/// Returns last zone index that can be found between start and end position, direction according windows ascending
/// REMARK: Size of area to be checked has influence to performance of method
METHOD M_GetLastZoneIndex : UINT // Returns ZoneIndex > 0, otherwise 0
VAR_INPUT
	mAbsoluteStartPosition	: UDINT; // Start position on the tracking [mm]
	mAbsoluteEndPosition	: UDINT; // End position on the tracking [mm]
	mOnlyZonesWithTU		: BOOL; // Check only zones with physical TU
END_VAR
END_METHOD

/// Searches through all available zones and add all zone index of ActionId to pData
/// Remark: Amount of available zones has influence to performance.
/// Remark: Existing entries in pData get overwritten.
METHOD M_GetPendingAssignments : BOOL // Returns true if all found zones could be added to pData, otherwise false
VAR_INPUT
	mActionId				: INT; // ID of action which requests zone (<>0)
	mpData 					: POINTER TO UINT; // Address of Value or Array to store the result
	mDataLen				: UINT; // Size of data
END_VAR
VAR_OUTPUT
	mCount					: UINT; // Number of entries added to pData
END_VAR
END_METHOD

/// Converts an absolute position into the current position on the tracking
METHOD M_GetTrackingPosition : UDINT // Converted position on tracking [mm]
VAR_INPUT
	mAbsolutePosition	: UDINT; // Absolute position 
END_VAR
END_METHOD

/// Returns TU end position of a zone on tracked distance
/// Remark: When no TU available the return value is 0, but is notfied with output "NoTuAvailable"
METHOD M_GetTU_EndPosition : UDINT // Returns position of TU end [mm]
VAR_INPUT
	mZoneIndex			: UINT; // Index of zone
END_VAR
VAR_OUTPUT
	mNoTU_Available		: BOOL; // No TU Available
END_VAR
END_METHOD

/// Returns TU start position of a zone on tracked distance
/// Remark: When no TU available the return value is 0, but is notfied with output "NoTuAvailable"
METHOD M_GetTU_StartPosition : UDINT // Start position of TU [mm]
VAR_INPUT
	mZoneIndex			: UINT; // Index of zone
END_VAR
VAR_OUTPUT
	mNoTU_Available		: BOOL; // No TU Available
END_VAR
END_METHOD

/// Returns position of Zone end on tracked distance
METHOD M_GetZoneEndPosition : UDINT // Position of Zone end [mm]
VAR_INPUT
	mZoneIndex			: UINT; // Index of zone
END_VAR
END_METHOD

/// Returns ZoneIndex at AbsolutePosition
METHOD M_GetZoneIndex : UINT // Returns ZoneIndex > 0, otherwise 0
VAR_INPUT
	mAbsolutePosition	: UDINT; // Position on the tracking [mm]
END_VAR
END_METHOD

/// Returns position of Zone start on tracked distance
METHOD M_GetZoneStartPosition : UDINT // Position of Zone start [mm]
VAR_INPUT
	mZoneIndex			: UINT; // Index of zone
END_VAR
END_METHOD

/// Inhibits shifting on a specific zone
METHOD M_InhibitShifting : BOOL // Returns true if successfully, otherwise false (e.g. Zone not found or not in use)
VAR_INPUT
	mZoneIndex		: UINT; // Zone index
	mInhibit		: BOOL; // True = Inhibit shifting
END_VAR
END_METHOD

/// Checks if a TU or a part of it, is found in a certain range.
METHOD M_IsTU_InRange : BOOL; // Returns true if present, otherwise false
VAR_INPUT
	mZoneIndex				: UINT; // Tracking zone index
	mAbsoluteStartRange		: UDINT; // Start range position on the tracking [mm]
	mAbsoluteEndRange		: UDINT; // End range position on the tracking [mm]
END_VAR
END_METHOD

/// Returns if a physical TU is present at mAbsolutePosition
METHOD M_IsTU_Present : BOOL; // Returns true if present, otherwise false
VAR_INPUT
	mAbsolutePosition		: UDINT; // Absolute position on tracking length
END_VAR
END_METHOD

/// Checks if a zone or a part of it,  is found in a certain range.
METHOD M_IsZoneInRange : BOOL; // Returns true if zone is in range, otherwise false
VAR_INPUT
	mZoneIndex				: UINT; // Tracking zone index
	mAbsoluteStartRange		: UDINT; // Start range position on the tracking [mm]
	mAbsoluteEndRange		: UDINT; // End range position on the tracking [mm]
END_VAR
END_METHOD

/// This function synchronize only a Front edge to a specific position and calculates the new TU length.
/// Remark: Zone begin gets adjusted to new front edge position. Spare windows in front of front edge get removed.
/// Remark: If at absolute position no zone is found, it search to the left for next front edge
/// until "mMaxFrontEdgeDeviation" to find one to synchronize.
METHOD M_ResyncOnlyFE : UINT // Returns > 0 of the synchronized Zone index, otherwise 0 (e.g. No Zone, No occupied zone)
VAR_INPUT
	mAbsolutePosition		: UDINT; // Absolute position [mm]
	mMaxFrontEdgeDeviation 	: UDINT; (* When zone can not be found at "Absolute position",
										a search upwards is executed to a limit of MaxFrontEdgeDeviation [mm]*)
END_VAR
END_METHOD

/// This function synchronize only Rear edge to a specific position and calculates new TU length.
/// Remark: Zone end gets adjusted to new rear edge position. Spare windows after rear edge get removed.
/// Remark: If at absolute position no zone is found, it search to the right
/// until "mMaxFrontEdgeDeviation" to find one to synchronize.
METHOD M_ResyncOnlyRE : UINT // Returns > 0 of the synchronized Zone index, otherwise 0
VAR_INPUT
	mAbsolutePosition		: UDINT; // Absolute position [mm]
	mMaxRearEdgeDeviation 	: UDINT; (* When zone can not be found at "Absolute position",
										a search upwards is executed to a limit of MaxRearEdgeDeviation [mm]*)
END_VAR
END_METHOD

/// This function synchronize whole TU aligned by Front edge to a specific position.
/// Rear edge is adjusted automatically to keep the length of TU.
/// Remark: If at absolute position no zone is found, it search to the left
/// until "mMaxFrontEdgeDeviation" to find one to synchronize.
METHOD M_ResyncTU_FE : UINT // Returns > 0 of the synchronized Zone index, otherwise 0
VAR_INPUT
	mAbsolutePosition		: UDINT; // Absolute position [mm]
	mMaxFrontEdgeDeviation 	: UDINT; (* When zone can not be found at "Absolute position",
										a search upwards is executed to a limit of MaxFrontEdgeDeviation [mm]*)
END_VAR
END_METHOD

/// This function synchronize whole TU aligned by Rear edge to a specific position.
/// Front edge is adjusted automatically to keep the length of TU.
/// Remark: If at absolute position no zone is found, it search to the right
/// until "mMaxFrontEdgeDeviation" to find one to synchronize.
METHOD M_ResyncTU_RE : UINT // Returns > 0 of the synchronized Zone index, otherwise 0
VAR_INPUT
	mAbsolutePosition		: UDINT; // Absolute position [mm]
	mMaxRearEdgeDeviation 	: UDINT; (* When zone can not be found at "Absolute position",
										a search upwards is executed to a limit of MaxRearEdgeDeviation [mm]*)
END_VAR
END_METHOD

/// Enlarges a zone by given value to upstream direction
METHOD M_ShortenZone : BOOL
VAR_INPUT
	mZoneIndex 				: UINT; // Zone index to enlarge
	mReductionLength		: UINT; // Reduce existing zone by this length [mm]
	mShiftFrontEdge			: BOOL; // Shift front edge for reduction
END_VAR
END_METHOD

/// Returns currently available amount of TUs
PROPERTY P_TU_Count : INT
GET
END_GET
END_PROPERTY

/// Access to Window table  for read operations
/// Remark: User has to ensure that writing does not influence the process in a bad way.
{attribute 'suppress_wrn_C0410'}
PROPERTY P_WindowTable : REFERENCE TO ARRAY[1..WindowTracking.MAX_NUMBER_OF_WINDOWS] OF ST_WindowTrackingWindow;
GET
END_GET
END_PROPERTY

/// Returns currently available amount of Zones
PROPERTY P_ZoneCount : INT
GET
END_GET
END_PROPERTY

/// Access to Zone table  for read operations
/// Remark: User has to ensure that writing does not influence the process in a bad way.
{attribute 'suppress_wrn_C0410'}
PROPERTY P_ZoneTable : REFERENCE TO ARRAY[1..WindowTracking.MAX_NUMBER_OF_ZONES] OF ST_WindowTrackingZone;
GET
END_GET
END_PROPERTY

END_INTERFACE

// ---- 20_Product/30_Toolbox/17_WindowTracking/10_Core/02_ITFs/I_WindowTrackingListener.TcIO
/// Window tracking listener 
INTERFACE I_WindowTrackingListener EXTENDS __System.IQueryInterface

/// Shifting completed event
METHOD M_TrackingShiftingCompletedEvent
VAR_INPUT
	mAbsolutePosition		: UDINT; // Absolute shifting start position [mm]
	mDistance				: UDINT; // Distance [mm] to be shifted
	mWindowIndex			: UINT; // Absolute position as window index on tracking
	mWindowsToShift			: UINT; // Distance to be shifted in amount of windows
END_VAR
END_METHOD

/// Shifting initiated event
METHOD M_TrackingShiftingInitiatedEvent
VAR_INPUT
	mAbsolutePosition		: UDINT; // Absolute shifting start position [mm]
	mDistance				: UDINT; // Distance [mm] to be shifted
	mWindowIndex			: UINT; // Absolute position as window index on tracking
	mWindowsToShift			: UINT; // Distance to be shifted in amount of windows
END_VAR
END_METHOD

/// Window tracking allocated new zone
METHOD M_TrackingTU_AddedEvent
VAR_INPUT
	mTrackingZoneIndex	: UINT; // New Zone index 
	mTrackingZoneData	: ST_WindowTrackingZone; // Data of deleted zone
END_VAR
END_METHOD

/// Window tracking deleted this zone
METHOD M_TrackingTU_DeletedEvent
VAR_INPUT
	mTrackingZoneIndex	: UINT; // Deleted zone index
	mTrackingZoneData	: ST_WindowTrackingZone; // Data of deleted zone
END_VAR
END_METHOD

/// Window tracking allocated new zone
METHOD M_TrackingZoneAddedEvent
VAR_INPUT
	mTrackingZoneIndex	: UINT; // New Zone index 
	mTrackingZoneData	: ST_WindowTrackingZone; // Data of deleted zone
END_VAR
END_METHOD

/// Window tracking deleted this zone
METHOD M_TrackingZoneDeletedEvent
VAR_INPUT
	mTrackingZoneIndex	: UINT; // Deleted zone index
	mTrackingZoneData	: ST_WindowTrackingZone; // Data of deleted zone
END_VAR
END_METHOD

/// A zone was enlarged event
METHOD M_TrackingZoneEnlargedEvent
VAR_INPUT
	mTrackingZoneIndex	: UINT; // Enlarged Zone index 
END_VAR
VAR_IN_OUT
	mOldTrackingZoneData : ST_WindowTrackingZone; // Zone data before modification
	mNewTrackingZoneData : ST_WindowTrackingZone; // Zone data after modification
END_VAR
END_METHOD

/// Window tracking moved this zone
METHOD M_TrackingZoneMovedEvent
VAR_INPUT
	mTrackingZoneIndex	: UINT; // Deleted zone index
	mTrackingZoneData	: ST_WindowTrackingZone; // Data of deleted zone
END_VAR
END_METHOD

/// A zone was shortened event
METHOD M_TrackingZoneShortenedEvent
VAR_INPUT
	mTrackingZoneIndex	: UINT; // Shortened Zone index 
END_VAR
VAR_IN_OUT
	mOldTrackingZoneData : ST_WindowTrackingZone; // Zone data before modification
	mNewTrackingZoneData : ST_WindowTrackingZone; // Zone data after modification
END_VAR
END_METHOD

END_INTERFACE

// ---- 20_Product/20_ProBox/MainProBox.TcPOU
PROGRAM MainProBox
(**************************************************************************************
 * 	Application		:	ProBox
 *	Revision		:	$$
 *	Revision date	:	$$
 *	Last changed by	:	$$
 *	URL				:	$$
 *
 *	Purpose			:	ProBox main application.
 *
 * ------------------------------------------------------------------------------------
 *	Copyright Swisslog [IP AG], Switzerland. All rights reserved.
 * 
 * ------------------------------------------------------------------------------------
 *	
 * 	Revision History: 
 *
 * 	VERSION			DATE			INITIALS			DESCRIPTION
 *	0.1				01.01.2001		swl					Example
 *
 **************************************************************************************)
VAR
	fbHardwareInputs					: FB_HardwareInputs;
	fbHardwareOutputs					: FB_HardwareOutputs;	
	fbSafetyCustomization				: FB_SafetyCompositionCustomized;
END_VAR
VAR_TEMP
BCFisInitiaded:BOOL;
		
END_VAR

 
(***************************************************************************************************************
  
***************************************************************************************************************)
BCFisInitiaded :=MainConv.Init;

EMULATION_ENABLED := TRUE;
IF(EMULATION_ENABLED) THEN
	MainConvEmulation();
END_IF

IF(BCFisInitiaded) THEN 
	IF(NOT EMULATION_ENABLED) THEN
		// Get HW Inputs
		fbHardwareInputs();
	END_IF		
	// run Custom debug functions
	F_DebugCompositionCustomization();  
END_IF
	
// Custom safety functions 
fbSafetyCustomization(_InitSafety:=BCFisInitiaded AND NOT EMULATION_ENABLED);
//run BCF
MainConv();

//if MainConv is initiated and not emulation enabled
IF(BCFisInitiaded) THEN
	//Set HW Outputs
	fbHardwareOutputs();		
END_IF

END_PROGRAM

// ---- 10_Project/10_App/11_Custom/FB_HardwareInputs.TcPOU
FUNCTION_BLOCK FB_HardwareInputs


;
// Example
(*
fbSG_001.HW_Inputs 								:= I_11_001_SG;
fbSG_001.HW_Inputs.ResetErrorPB 				:= I_11_001_SG.AutoOnPB;
fbSG_001.HW_Inputs.FeedbackMainContactorOFF[4] 	:= FALSE;
fbSG_001.HW_Inputs.EmergencyCircuitOK 			:= TRUE;
fbSG_001.HW_Inputs.MainContactorOFF 			:= I_11_001_SG.MainContactorOFF;

Main_Contactor_ON_Q := Main_Contactor_ON_I;
Main_Contactor_OFF_Q := Main_Contactor_OFF_I;
*)

END_FUNCTION_BLOCK

// ---- 10_Project/10_App/11_Custom/FB_HardwareOutputs.TcPOU
FUNCTION_BLOCK FB_HardwareOutputs


;
// Example
(*
Q_11_001_SG := fbSG_001.HW_Outputs;
Q_11_001_SG_Beacon_Error := fbSG_001.HW_Outputs.ErrorPending;
Q_11_001_SG_Beacon_Auto := fbSG_001.HW_Outputs.GroupStarted;
*)

END_FUNCTION_BLOCK

// ---- 10_Project/10_App/11_Custom/FB_SafetyCompositionCustomized.TcPOU
FUNCTION_BLOCK FB_SafetyCompositionCustomized
VAR_INPUT
	///true if initializing is active
	_InitSafety: BOOL;
END_VAR


IF(_InitSafety) Then
	//Add project specific safety code that shall execute during PLC init/reinit. 
	;
ELSE
	//Add project specific safety code here. 
	//renamed from Com_Error to FB_SafetyCompositionCustomized
	;
END_IF

END_FUNCTION_BLOCK

// ---- 20_Product/10_BCF/11_Conv/MainConv.TcPOU
PROGRAM MainConv
(**************************************************************************************
 * 	Application		:	BoxControl Framework
 *	Revision		:	$Revision: 404529 $
 *	Revision date	:	$Date: 2018-04-23 08:21:38 +0200 (Mo., 23 Apr 2018) $
 *	Last changed by	:	$Author: b7bolm $
 *	URL				:	$URL: http://almscdc.swisslog.com/repo/SWPD/Development/BoxControlFramework/20_Release/trunk/01_Software/BCF/BCF/JumpStart/20_Product/10_App/MainConv.TcPOU $
 *
 *	Purpose			:	Main program call.
 *
 * ------------------------------------------------------------------------------------
 *	Copyright Swisslog [IP AG], Switzerland. All rights reserved.
 * 
 * ------------------------------------------------------------------------------------
 *	
 * 	Revision History: 
 *
 * 	VERSION			DATE			INITIALS			DESCRIPTION
 *	0.1				01.01.2001		swl					Example
  *
 **************************************************************************************)
VAR
	Init								: BOOL := FALSE; // Application is initialized 
	
	ActivateSubsystemConfig				: BOOL; // Flag to activate the configuration of the Subsystem 
	ActivateGroupManagerConfig			: BOOL; // Flag to activate the configuration of the groupmanager 
	ActivateGroupConfig					: BOOL; // Flag to activate the configuration of the group 
	ActivatePositionConfig				: BOOL; // Flag to activate the configuration of the element 
	ActivateCommunicationConfig			: BOOL; // Flag to activate the configuration of the communication 
	
	InitializeSubsystem					: BOOL; // Flag to activate initialization
	InitializeGroupManager				: BOOL; // Flag to activate initialization
	InitializeGroups					: BOOL; // Flag to activate initialization
	InitializeFunctions					: BOOL; // Flag to activate initialization
	InitializeCommunication				: BOOL; // Flag to activate initialization
	InitializeElements					: BOOL; // Flag to activate initialization
	ReInit								: BOOL := TRUE; // Reinitialize application
	fbDebugMsg							: FB_DebugMsg; // Debug instance
	fbGetSystemTime						: GETSYSTEMTIME; // Gets the system time  
	LatchedTimeDW						: DWORD; // Latch the system time 
	LastTimeStamp						: DWORD; // Time stamp
	fbGetCurTaskIdx  					: GETCURTASKINDEX; // Returns the actual task index
	
	fbCommunicationComposition			: FB_CommunicationComposition; // Communication call
	fbElementComposition				: FB_ElementComposition; // Element calls
	fbElementCompositionCustomized		: FB_ElementCompositionCustomized; // Element calls
	fbFunctionComposition				: FB_FunctionComposition; // Function calls
	fbFunctionCompositionCustomized		: FB_FunctionCompositionCustomized; // Function calls
	fbGroupComposition					: FB_GroupComposition; // Group calls
	fbGroupCompositionCustomized		: FB_GroupCompositionCustomized; // Group calls
	fbSubsystemComposition				: FB_SubsystemComposition; // Subsystem calls
	fbSubsystemCompositionCustomized	: FB_SubsystemCompositionCustomized; // Subsystem calls
	fbDeleteOldTU_Data					: FB_DeleteOldTU_Data; // Checks old TU data
	SubsystemState						: ST_PositionState; // Subsystem state
END_VAR

// whow

(**************************************************************************************************************
   Update PLC data
***************************************************************************************************************)
A_UpdatePLC_Data();

(**************************************************************************************************************
   Detect PLC restart
***************************************************************************************************************)
A_DetectPLC_Restart();

(**************************************************************************************************************
   Initialize program
***************************************************************************************************************)
A_Init();

(**************************************************************************************************************
   Call global instances
***************************************************************************************************************)
A_GlobalInstances();

(**************************************************************************************************************
   Call application
***************************************************************************************************************)
IF Init THEN

	(**************************************************************************************************************
	   Update all references
	***************************************************************************************************************)
	F_UpdateReferences();

	(**************************************************************************************************************
	   Update all ISR signals
	***************************************************************************************************************)
	F_UpdateISR();
	
	(**************************************************************************************************************
	   Clean up TU-Data table
	***************************************************************************************************************)
	A_DeleteOldTU_Data();

	(**************************************************************************************************************
	  Call functional units
	***************************************************************************************************************)
	// Communication 
	fbCommunicationComposition();

	// Subsystem
	fbSubsystemCompositionCustomized();
	fbSubsystemComposition();

	// Groups
	fbGroupCompositionCustomized();
	fbGroupComposition();
	
	// Elements 
	fbElementCompositionCustomized();
 	fbElementComposition();
			
	// Functions
	fbFunctionCompositionCustomized();
	fbFunctionComposition();

	// Call supplements (e.g. Commissioning tools)
	A_Supplements();

END_IF

ACTION A_DeleteOldTU_Data:
(**************************************************************************************
 * 	NAME		A_DeleteOldTU_Data
 * 	FUNCTION	Delete old TU data
 **************************************************************************************)
// Get subsystem state
SubsystemState := F_GetSubsystemOperationState();

// Subsystem is started
IF SubsystemState.eState = E_PositionState.STARTED THEN

	// Check old TU data
	fbDeleteOldTU_Data();
END_IF
END_ACTION

ACTION A_DetectPLC_Restart:
(**************************************************************************************
 * 	NAME		A_DetectPLC_Restart
 * 	FUNCTION	Detects a PLC restart
 **************************************************************************************)

// Get current cycle count
fbGetCurTaskIdx();

// Get Timestamp
IF LatchedTimeDW <= fbGetSystemTime.timeLoDW THEN
	// No overflow 
	IF ((fbGetSystemTime.timeLoDW - LatchedTimeDW) > 10 * _TaskInfo[fbGetCurTaskIdx.index].CycleTime )THEN
		// PLC was stopped reactivate start delay -> Reinit
		ReInit := TRUE;
	END_IF
ELSE
	// Overflow hapened
	IF ((fbGetSystemTime.timeLoDW + (4294967296- LatchedTimeDW)) > 10 * _TaskInfo[fbGetCurTaskIdx.index].CycleTime) THEN
		// PLC was stopped reactivate start delay -> Reinit
		ReInit := TRUE;
	END_IF
END_IF

// Update latched time
LatchedTimeDW := fbGetSystemTime.timeLoDW;
END_ACTION

ACTION A_GlobalInstances:
(**************************************************************************************
 * 	NAME		A_GlobalInstances
 * 	FUNCTION	Call global instances
 **************************************************************************************)

// Call blink pulses
fbBlink_1s();
fbBlink_100ms();
fbBlink_500ms();
END_ACTION

ACTION A_Init:
(**************************************************************************************
 * 	NAME		A_Init
 * 	FUNCTION	Initialize application
 **************************************************************************************)
// Reset socket closer
fbSocketCloseAll(bExecute:= FALSE);	

// Force reinitialization
IF ReInit THEN
	(*
	As a reason that it possible that the application
	was NOT stopped properly, all socket connections
	need to be closed during init
	*)
	System.fbSocketCloseAll(bExecute:= TRUE);	
	// Force init of application
	Init := FALSE;
	// Reset values
	ReInit := FALSE; 
END_IF

(*
	Initialize the application if socket close is done, and
	we have a system time available
*)
IF NOT Init AND NOT fbSocketCloseAll.bBusy AND fbSystemTime.TIMESTR.wYear > 0 THEN
	Init := TRUE;

	// Update all references before using them after a reset 
	F_UpdateReferences();
	
	// Load configurations
	F_ConfigProduct();
	F_ConfigCommunication();
	F_ConfigPosition();
	F_ConfigGroup();
	F_ConfigGroupManager();
	F_ConfigSubsystem();
	F_ConfigExternalDestination();

	(* 
	The initialization order should not be changed!
	Changing this order can lead to undexpected behavior, 
	or inconsisten data values
	*)	
	F_InitializeCommunication();
	
	// Force init Subsystem
	F_InitializeSubsystem();
	
	// Force initializing Group manager 
	fbGroupManager.M_Init(TRUE);

	// Initialize all groups
	F_InitializeAllGroups();
	
	// Initialize all elements
	F_InitializeAllElements();
	
	// Initialize all functions
	F_InitializeAllFunctions();

	fbDebugMsg.M_SendInfoMsg('Main initialized.');
END_IF
END_ACTION

ACTION A_Supplements:
(**************************************************************************************
 * 	NAME		A_Supplements
 * 	FUNCTION	Help functionalities - E.g. commissioning tools, functions...
 **************************************************************************************)

// Load communication configuration, only used for commissioning 
IF ActivateCommunicationConfig THEN
	F_ConfigCommunication();
	ActivateCommunicationConfig := FALSE;
END_IF

// Load position configuration, only used for commissioning 
IF ActivatePositionConfig THEN
	F_ConfigPosition();
	ActivatePositionConfig := FALSE;
END_IF

// Load group configuration, only used for commissioning 
IF ActivateGroupConfig THEN
	F_ConfigGroup();
	ActivateGroupConfig := FALSE;
END_IF

// Load groupmanager configuration, only used for commissioning 
IF ActivateGroupManagerConfig THEN
	F_ConfigGroupManager();
	ActivateGroupManagerConfig := FALSE;
END_IF

// Load Subsystem configuration, only used for commissioning 
IF ActivateSubsystemConfig THEN
	F_ConfigSubsystem();
	ActivateSubsystemConfig := FALSE;
END_IF

// Force init
IF InitializeSubsystem THEN
	InitializeSubsystem := FALSE;
	// Force init Subsystem
	F_InitializeSubsystem();
END_IF

// Force init
IF InitializeGroupManager THEN
	InitializeGroupManager := FALSE;
	// Force initializing Group manager 
	fbGroupManager.M_Init(TRUE);
END_IF	
	
// Force init
IF InitializeGroups THEN
	InitializeGroups := FALSE;
	// Initialize all groups
	F_InitializeAllGroups();
END_IF	

// Force init
IF InitializeFunctions THEN
	InitializeFunctions := FALSE;
	// Initialize all funcitons
	F_InitializeAllFunctions();
END_IF		

// Force init
IF InitializeElements THEN
	InitializeElements := FALSE;
	// Initialize all elements
	F_InitializeAllElements();
END_IF	

// Force init
IF InitializeCommunication THEN
	InitializeCommunication := FALSE;
	// Close all connections
	F_InitializeCommunication();
END_IF
END_ACTION

ACTION A_UpdatePLC_Data:
(**************************************************************************************
 * 	NAME		A_UpdatePLC_Data
 * 	FUNCTION	Updates all PLC data variables
 **************************************************************************************)

// System time
fbSystemTime(START:= TRUE);
IF NOT fbSystemTime.BUSY THEN
	// not busy anymore -> restart
	fbSystemTime(START:= FALSE);
	fbSystemTime(START:= TRUE);
END_IF


// Save system time in global variable
TimeStampDT    := SYSTEMTIME_TO_DT    (fbSystemTime.TIMESTR);
TimeStampString:= SYSTEMTIME_TO_STRING(fbSystemTime.TIMESTR);


// Get System Time
fbGetSystemTime();

// Get Cycle Time
IF fbGetSystemTime.timeLoDW > LastTimeStamp THEN
	ActCycleTime := UDINT_TO_DINT((fbGetSystemTime.timeLoDW - LastTimeStamp + 5) / 10);
END_IF

// Update last time stamp
LastTimeStamp := fbGetSystemTime.timeLoDW;
END_ACTION

END_PROGRAM

// ---- 20_Product/10_BCF/10_Base/11_Com/12_DebugMsg/FB_DebugMsg.TcPOU
{attribute 'reflection'}
FUNCTION_BLOCK FB_DebugMsg
(**************************************************************************************
 * 	Application		:	BoxControl Framework
 *	Revision		:	$Revision: 404529 $
 *	Revision date	:	$Date: 2018-04-23 08:21:38 +0200 (Mo., 23 Apr 2018) $
 *	Last changed by	:	$Author: b7bolm $
 *	URL				:	$URL: http://almscdc.swisslog.com/repo/SWPD/Development/BoxControlFramework/20_Release/trunk/01_Software/BCF/BCF/JumpStart/20_Product/10_App/11_Com/10_Lib/FB_DebugMsg.TcPOU $
 *
 *	Purpose			:	Debug massage
 *
 * ------------------------------------------------------------------------------------
 *	Copyright Swisslog [IP AG], Switzerland. All rights reserved.
 * 
 * ------------------------------------------------------------------------------------
 *	
 * 	Revision History: 
 *
 * VERSION DATE         INITIALS     DESCRIPTION
 * 0.0     DD.MM.YYYY   (name)       (explain customized modifications)
 *
 **************************************************************************************)
VAR
	{attribute 'instance-path'}
	{attribute 'no_init'}
	InstanceName				: STRING[System.DEBUGSOURCELENGTH];
	//------------------------------------------------------------------
	LastMessage					: STRING[System.DEBUGMESSAGELENGTH];
	fbGetCurTaskIdx				: GETCURTASKINDEX; // Returns the actual task index
	LastCycleCounterValue		: UDINT;
END_VAR

// Body never called

METHOD FB_init : BOOL

(********************************************************************************************************************************)
VAR_INPUT
	bInitRetains          : BOOL; // if TRUE, the retain variables are initialized (warm start / cold start)
	bInCopyCode           : BOOL;  // if TRUE, the instance afterwards gets moved into the copy code (online change)
  (*----------------------------------------------------------------------------------------------------------------------------*)
END_VAR

(********************************************************************************************************************************)
VAR
END_VAR

(********************************************************************************************************************************)
(** remove 'QB2Jumpstart.JumpStart.' from instance path *************************************************************************)
F_InstancePathRemovals(DestStart     := ADR(InstanceName),
                       DestEnd       := ADR(InstanceName) + SIZEOF(InstanceName),
                       RemoveLastPart:= TRUE);  




(********************************************************************************************************************************)
(** done ************************************************************************************************************************)
END_METHOD

METHOD M_SendErrorMsg
(**************************************************************************************
 * 	Application		:	BoxControl Framework
 *	Revision		:	$Revision: 404529 $
 *	Revision date	:	$Date: 2018-04-23 08:21:38 +0200 (Mo., 23 Apr 2018) $
 *	Last changed by	:	$Author: b7bolm $
 *	URL				:	$URL: http://almscdc.swisslog.com/repo/SWPD/Development/BoxControlFramework/20_Release/trunk/01_Software/BCF/BCF/JumpStart/20_Product/10_App/11_Com/10_Lib/FB_DebugMsg.TcPOU $
 *
 *	Purpose			:	Send error message
 *
 * ------------------------------------------------------------------------------------
 *	Copyright Swisslog [IP AG], Switzerland. All rights reserved.
 * 
 * ------------------------------------------------------------------------------------
 *	
 * 	Revision History: 
 *
 * 	VERSION			DATE			INITIALS			DESCRIPTION
 *	0.1				01.01.2001		swl					Example
 *
 **************************************************************************************)
VAR_INPUT
	mMessage	: STRING(System.DEBUGMESSAGELENGTH);
END_VAR
// message is not equal to last sent message
// same message can be sent in same cycle several times
fbDebugMsgManager.M_SendMessage(E_DebugMsgType.ERROR, InstanceName, ADR(mMessage), INT_TO_UDINT(LEN(mMessage)));
LastMessage := mMessage;
// Get current cycle count
fbGetCurTaskIdx();
LastCycleCounterValue := _TaskInfo[fbGetCurTaskIdx.index].CycleCount;
END_METHOD

METHOD M_SendInfoMsg
(**************************************************************************************
 * 	Application		:	BoxControl Framework
 *	Revision		:	$Revision: 404529 $
 *	Revision date	:	$Date: 2018-04-23 08:21:38 +0200 (Mo., 23 Apr 2018) $
 *	Last changed by	:	$Author: b7bolm $
 *	URL				:	$URL: http://almscdc.swisslog.com/repo/SWPD/Development/BoxControlFramework/20_Release/trunk/01_Software/BCF/BCF/JumpStart/20_Product/10_App/11_Com/10_Lib/FB_DebugMsg.TcPOU $
 *
 *	Purpose			:	Send info message
 *
 * ------------------------------------------------------------------------------------
 *	Copyright Swisslog [IP AG], Switzerland. All rights reserved.
 * 
 * ------------------------------------------------------------------------------------
 *	
 * 	Revision History: 
 *
 * 	VERSION			DATE			INITIALS			DESCRIPTION
 *	0.1				01.01.2001		swl					Example
 *
 **************************************************************************************)
VAR_INPUT
	mMessage			: STRING(System.DEBUGMESSAGELENGTH);
END_VAR
// message is not equal to last sent message
// same message can be sent in same cycle several times
fbDebugMsgManager.M_SendMessage(E_DebugMsgType.INFO, InstanceName, ADR(mMessage), INT_TO_UDINT(LEN(mMessage)));
LastMessage := mMessage;
// Get current cycle count
fbGetCurTaskIdx();
LastCycleCounterValue := _TaskInfo[fbGetCurTaskIdx.index].CycleCount;
END_METHOD

METHOD M_SendLongMsg
(**************************************************************************************
 * 	Application		:	BoxControl Framework
 *	Revision		:	$Revision: 404529 $
 *	Revision date	:	$Date: 2018-04-23 08:21:38 +0200 (Mo., 23 Apr 2018) $
 *	Last changed by	:	$Author: b7bolm $
 *	URL				:	$URL: http://almscdc.swisslog.com/repo/SWPD/Development/BoxControlFramework/20_Release/trunk/01_Software/BCF/BCF/JumpStart/20_Product/10_App/11_Com/10_Lib/FB_DebugMsg.TcPOU $
 *
 *	Purpose			:	Send long message
 *						Long messages will be separated in messages < MAX_STRING_LENGTH
 *						and forwarded as normal messages.
 *
 * ------------------------------------------------------------------------------------
 *	Copyright Swisslog [IP AG], Switzerland. All rights reserved.
 * 
 * ------------------------------------------------------------------------------------
 *	
 * 	Revision History: 
 *
 * 	VERSION			DATE			INITIALS			DESCRIPTION
 *	0.1				01.01.2001		swl					Example
 *
 **************************************************************************************)
VAR_INPUT
	mDebugMsgType	: E_DebugMsgType; // Message type
	mpData			: PVOID; // Address to data source
	mLen			: UDINT; // Length of the message (Attention, if the input is String use LEN instead of SIZEOF
END_VAR

// message is not equal to last sent message
// same message can be sent in same cycle several times
fbDebugMsgManager.M_SendMessage(mDebugMsgType, InstanceName, mpData, mLen);

// Store first 255 characters for debugging
F_BlockCopy(
	pSrc:= mpData, 
	LenSrc:= mLen, 
	pDest:= ADR(LastMessage), 
	LenDest:= SIZEOF(LastMessage));
	
// Get current cycle count
fbGetCurTaskIdx();
LastCycleCounterValue := _TaskInfo[fbGetCurTaskIdx.index].CycleCount;
END_METHOD

METHOD M_SendWarningMsg
(**************************************************************************************
 * 	Application		:	BoxControl Framework
 *	Revision		:	$Revision: 404529 $
 *	Revision date	:	$Date: 2018-04-23 08:21:38 +0200 (Mo., 23 Apr 2018) $
 *	Last changed by	:	$Author: b7bolm $
 *	URL				:	$URL: http://almscdc.swisslog.com/repo/SWPD/Development/BoxControlFramework/20_Release/trunk/01_Software/BCF/BCF/JumpStart/20_Product/10_App/11_Com/10_Lib/FB_DebugMsg.TcPOU $
 *
 *	Purpose			:	Send warning message
 *
 * ------------------------------------------------------------------------------------
 *	Copyright Swisslog [IP AG], Switzerland. All rights reserved.
 * 
 * ------------------------------------------------------------------------------------
 *	
 * 	Revision History: 
 *
 * 	VERSION			DATE			INITIALS			DESCRIPTION
 *	0.1				01.01.2001		swl					Example
 *
 **************************************************************************************)
VAR_INPUT
	mMessage		: STRING(System.DEBUGMESSAGELENGTH);
END_VAR
// message is not equal to last sent message
// same message can be sent in same cycle several times
fbDebugMsgManager.M_SendMessage(E_DebugMsgType.WARNING, InstanceName, ADR(mMessage), INT_TO_UDINT(LEN(mMessage)));
LastMessage := mMessage;
// Get current cycle count
fbGetCurTaskIdx();
LastCycleCounterValue := _TaskInfo[fbGetCurTaskIdx.index].CycleCount;;
END_METHOD

END_FUNCTION_BLOCK

// ---- 20_Product/10_BCF/10_Base/11_Com/01_Stringhandling/F_InstancePathRemovals.TcPOU
// removes 'QB2Jumpstart.JumpStart.' from instance path and if RemoveLastPart true, also last part '.yyyyy'
FUNCTION PUBLIC F_InstancePathRemovals

(**************************************************************************************
 * 	Application		:	BoxControl Framework
 *	Revision		  :	$Revision: 461868 $
 *	Revision date	:	$Date: 1979-01-09 14:35:13 +0200 (Di., 09 Jan 1979) $
 *	Last changed by	:	$Author: b7lipim $
 *	URL				:	$URL: http://almscdc.swisslog.com/repo/SWPD/Development/BoxControlFramework/20_Release/branches/R1.x/01_Software/BCF/BCF/JumpStart/20_Product/10_BCF/10_Base/11_Com/12_DebugMsg/00_GVLs/DebugTextBlocks.TcGVL $
 *
 * ------------------------------------------------------------------------------------
 *	Copyright Swisslog [IP AG], Switzerland. All rights reserved.
 * 
 * ------------------------------------------------------------------------------------
 *	
 * 	Revision History: 
 *
 * VERSION DATE         INITIALS     DESCRIPTION
 * 0.0     DD.MM.YYYY   (name)       (explain customized modifications)
 *
 **************************************************************************************)

(********************************************************************************************************************************)
VAR_INPUT
  DestStart             : POINTER TO BYTE                  := 0;     // = ADR(MyString)                    -> start position to concat
  DestEnd               : POINTER TO BYTE                  := 0;     // = ADR(MyString) + SIZEOF(MyString) -> buffer/string end
  (*----------------------------------------------------------------------------------------------------------------------------*)
  RemoveLastPart        : BOOL                             := FALSE; // also removes last (own) part
END_VAR

(********************************************************************************************************************************)
VAR
  Dest                  : POINTER TO BYTE                  := 0;
  Source                : POINTER TO BYTE                  := 0;
  End                   : POINTER TO BYTE                  := 0;
END_VAR



(********************************************************************************************************************************)
(** check inputs ****************************************************************************************************************)
IF   (DestStart = 0)         THEN  RETURN;
ELSIF(DestEnd   = 0)         THEN  RETURN;
ELSIF(DestStart >= DestEnd)  THEN  RETURN;
END_IF




(********************************************************************************************************************************)
(** remove 'QB2Jumpstart.JumpStart.' from instance path *************************************************************************)
Source:= DestStart;
(*-- first point ---------------------------------------------------------------------------------------------------------------*)
WHILE(Source^ <> 16#00)
DO
  // point found? -> store position ---------------------------------
  IF (Source^ = 16#2E)  (* '.' *)
  THEN
    Source:= Source + SIZEOF(Source^);
    EXIT;
  END_IF
  // next char ------------------------------------------------------
  Source:= Source + SIZEOF(Source^);
END_WHILE

(*-- second point --------------------------------------------------------------------------------------------------------------*)
WHILE(Source^ <> 16#00)
DO
  // point found? -> store position ---------------------------------
  IF (Source^ = 16#2E)  (* '.' *)
  THEN
    Source:= Source + SIZEOF(Source^);
    EXIT;
  END_IF
  // next char ------------------------------------------------------
  Source:= Source + SIZEOF(Source^);
END_WHILE




(********************************************************************************************************************************)
(** copying text ****************************************************************************************************************)
Dest:= DestStart;
WHILE(Source^ <> 16#00)
DO
  Dest^:= Source^;
  // point found? -> store position ---------------------------------
  IF (Dest^ = 16#2E)  (* '.' *)
  THEN
    End:= Dest;
  END_IF
  // next char ------------------------------------------------------
  Dest  := Dest   + SIZEOF(Dest^);
  Source:= Source + SIZEOF(Source^);
END_WHILE

Dest^:= 16#00;




(********************************************************************************************************************************)
(** remove also last part *******************************************************************************************************)
IF (RemoveLastPart = TRUE)
THEN
  IF (End <> 0)
  THEN
    End^:= 16#00;  // string ends at last found point
  END_IF
END_IF




(********************************************************************************************************************************)
(** done ************************************************************************************************************************)

END_FUNCTION

// ---- 20_Product/30_Toolbox/99_Misc/F_BlockCopy.TcPOU
FUNCTION F_BlockCopy : BOOL
VAR_INPUT
	pSrc	: PVOID;
	LenSrc  : UDINT;
	pDest 	: PVOID;
	LenDest	: UDINT;
END_VAR

VAR

END_VAR


IF LenSrc > 0 AND
   LenDest > 0 AND
   pSrc > 0 AND
   pDest > 0 THEN 
	
	MEMSET(destAddr := pDest, 0, LenDest);
   
	IF LenSrc > LenDest THEN	
		MEMCPY(destAddr := pDest, srcAddr := pSrc, n := LenDest);
	ELSE
		MEMCPY(destAddr := pDest, srcAddr := pSrc, n := LenSrc);
	END_IF

	F_BlockCopy := TRUE;
ELSE
	F_BlockCopy := FALSE;
END_IF

END_FUNCTION

// ---- 20_Product/10_BCF/11_Conv/10_Base/FB_CommunicationComposition.TcPOU
FUNCTION_BLOCK FB_CommunicationComposition
(**************************************************************************************
 * 	Application		:	BoxControl Framework
 *	Revision		:	$Revision: 404529 $
 *	Revision date	:	$Date: 2018-04-23 08:21:38 +0200 (Mo., 23 Apr 2018) $
 *	Last changed by	:	$Author: b7bolm $
 *	URL				:	$URL: http://almscdc.swisslog.com/repo/SWPD/Development/BoxControlFramework/20_Release/trunk/01_Software/BCF/BCF/JumpStart/20_Product/10_App/10_Base/10_Lib/10_Conv/FB_CommunicationComposition.TcPOU $
 *
 *	Purpose			:	Call communication composition
 *
 * ------------------------------------------------------------------------------------
 *	Copyright Swisslog [IP AG], Switzerland. All rights reserved.
 * 
 * ------------------------------------------------------------------------------------
 *	
 * 	Revision History: 
 *
 * 	VERSION			DATE			INITIALS			DESCRIPTION
 *	0.1				01.01.2001		swl					Example
 *
 **************************************************************************************)
VAR
	eMFCS_Channel			: E_MFCS_Channel; // Iterator MFCS channel
	MFCS_Instance			: ITF_MFCS; // Instance to compare valid interfaces
	StartTimeMeasurement	: T_DCTIME64;	// Get actual time stamp	
END_VAR


(**************************************************************************************************************
   Call all MFCS Channels   (e.g. SIS channels)
***************************************************************************************************************)
// Call all MFCS channels
FOR eMFCS_Channel := E_MFCS_Channel.BEGIN_CHANNEL + 1 TO E_MFCS_Channel.END_CHANNEL - 1 DO
	// Call communication service
	IF __QUERYINTERFACE(fbMFCS_Channel[eMFCS_Channel], MFCS_Instance) THEN
		// Start execution time measure
		StartTimeMeasurement := F_GetActualDcTime64();
		// Call communication service
		fbMFCS_Channel[eMFCS_Channel].M_CallCommunicationService();
		
		F_ExecutionTime(
			StartTime			:= StartTimeMeasurement,
			ExecutionTimeSlot 	:= ExecutionTimeTable.MFCS_Channels[eMFCS_Channel]);		
	END_IF
END_FOR

(**************************************************************************************************************
  Call the ITC message manager   
***************************************************************************************************************)
// Start execution time measure
StartTimeMeasurement := F_GetActualDcTime64();
// Call ITC service
fbITC_Manager.M_CallITC_Service();

F_ExecutionTime(
		StartTime			:= StartTimeMeasurement,
		ExecutionTimeSlot 	:= ExecutionTimeTable.ITC_Manager);

(**************************************************************************************************************
   Call the function block debug message manager  
***************************************************************************************************************)
// Start execution time measure
StartTimeMeasurement := F_GetActualDcTime64();
// Call
fbDebugMsgManager();

F_ExecutionTime(
		StartTime			:= StartTimeMeasurement,
		ExecutionTimeSlot 	:= ExecutionTimeTable.DebugMsgManager);

END_FUNCTION_BLOCK

// ---- 20_Product/10_BCF/10_Base/F_ExecutionTime.TcPOU
FUNCTION F_ExecutionTime : ULINT
(**************************************************************************************
 * 	Application		:	BoxControl Framework
 *	Revision		:	$Revision: 404529 $
 *	Revision date	:	$Date: 2018-04-23 08:21:38 +0200 (Mo., 23 Apr 2018) $
 *	Last changed by	:	$Author: b7bolm $
 *	URL				:	$URL: http://almscdc.swisslog.com/repo/SWPD/Development/BoxControlFramework/20_Release/trunk/01_Software/BCF/BCF/JumpStart/20_Product/10_App/10_Base/10_Lib/F_ExecutionTime.TcPOU $
 *
 *	Purpose			:	Measure execution time of a code section.
 *						This function reads out the current time value and build the 
 *						time difference to "StartTime" get the execution time.
 *						
 *						Measured in [ns]
 *
 * ------------------------------------------------------------------------------------
 *	Copyright Swisslog [IP AG], Switzerland. All rights reserved.
 * 
 * ------------------------------------------------------------------------------------
 *	
 * 	Revision History: 
 *
 * 	VERSION			DATE			INITIALS			DESCRIPTION
 *	0.1				01.01.2001		swl					Example
 *
 **************************************************************************************)
VAR_INPUT
	StartTime				: T_DCTIME64; // Start time	
END_VAR
VAR_IN_OUT
	ExecutionTimeSlot		: ST_ExecutionTime; // Execution time slot GVL: ExecutionTime
END_VAR
VAR
	CurrentTimeStamp		: T_DCTIME64;
END_VAR

// Get actual time stamp
CurrentTimeStamp := F_GetActualDcTime64();

IF StartTime > CurrentTimeStamp THEN
	// Overflow - skip measurement
	RETURN;
END_IF

// Calculate difference
ExecutionTimeSlot.CurrentValue := CurrentTimeStamp - StartTime;

// store max execution time
IF ExecutionTimeSlot.MaxValue < ExecutionTimeSlot.CurrentValue THEN
	ExecutionTimeSlot.MaxValue := ExecutionTimeSlot.CurrentValue;
END_IF

END_FUNCTION

// ---- 20_Product/10_BCF/11_Conv/10_Base/FB_ElementComposition.TcPOU
FUNCTION_BLOCK FB_ElementComposition
(**************************************************************************************
 * 	Application		:	BoxControl Framework
 *	Revision		:	$Revision: 404529 $
 *	Revision date	:	$Date: 2018-04-23 08:21:38 +0200 (Mo., 23 Apr 2018) $
 *	Last changed by	:	$Author: b7bolm $
 *	URL				:	$URL: http://almscdc.swisslog.com/repo/SWPD/Development/BoxControlFramework/20_Release/trunk/01_Software/BCF/BCF/JumpStart/20_Product/10_App/10_Base/10_Lib/10_Conv/FB_ElementComposition.TcPOU $
 *
 *	Purpose			:	Main program call.
 *
 * ------------------------------------------------------------------------------------
 *	Copyright Swisslog [IP AG], Switzerland. All rights reserved.
 * 
 * ------------------------------------------------------------------------------------
 *	
 * 	Revision History: 
 *
 * 	VERSION			DATE			INITIALS			DESCRIPTION
 *	0.1				01.01.2001		swl					Example
 *
 **************************************************************************************)
VAR
	eElementNumber		: E_ElementNumber; // Number of the element 
	fbDebugMsg			: FB_DebugMsg; // Debug Msg Manager (STACK) 
	DebugMsg			: T_MAXSTRING; // Debug msg
	StartTimeMeasurement: T_DCTIME64;	// Get actual time stamp
END_VAR

// Loop trough all elements 
FOR eElementNumber := E_BEGIN_ELEMENT + 1 TO E_END_ELEMENT - 1 DO
	// If this element is enabled 
	IF ElementRegistry[eElementNumber].Enable THEN
		// If a valid reference is available 
		IF __ISVALIDREF(ElementRegistry[eElementNumber].rElement) THEN
			// Start execution time measure
			StartTimeMeasurement := F_GetActualDcTime64();
			// Call
			ElementRegistry[eElementNumber].rElement();
			
			F_ExecutionTime(
				StartTime			:= StartTimeMeasurement,
				ExecutionTimeSlot 	:= ExecutionTimeTable.Elements[eElementNumber]);
		ELSE
			// Invalid reference
			DebugMsg := CONCAT('F_ElementComposition - Reference not valid, Element index: ', INT_TO_STRING(eElementNumber));
			fbDebugMsg.M_SendErrorMsg(mMessage := DebugMsg);
		END_IF
	END_IF
END_FOR

END_FUNCTION_BLOCK

// ---- 10_Project/10_App/11_Custom/FB_ElementCompositionCustomized.TcPOU
FUNCTION_BLOCK FB_ElementCompositionCustomized

;

END_FUNCTION_BLOCK

// ---- 20_Product/10_BCF/11_Conv/10_Base/FB_FunctionComposition.TcPOU
FUNCTION_BLOCK FB_FunctionComposition
(**************************************************************************************
 * 	Application		:	BoxControl Framework
 *	Revision		:	$Revision: 404529 $
 *	Revision date	:	$Date: 2018-04-23 08:21:38 +0200 (Mo., 23 Apr 2018) $
 *	Last changed by	:	$Author: b7bolm $
 *	URL				:	$URL: http://almscdc.swisslog.com/repo/SWPD/Development/BoxControlFramework/20_Release/trunk/01_Software/BCF/BCF/JumpStart/20_Product/10_App/10_Base/10_Lib/10_Conv/FB_FunctionComposition.TcPOU $
 *
 *	Purpose			:	Function call.
 *
 * ------------------------------------------------------------------------------------
 *	Copyright Swisslog [IP AG], Switzerland. All rights reserved.
 * 
 * ------------------------------------------------------------------------------------
 *	
 * 	Revision History: 
 *
 * 	VERSION			DATE			INITIALS			DESCRIPTION
 *	0.1				01.01.2001		swl					Example
 *
 **************************************************************************************)
VAR
	eFunctionNumber		: E_FunctionNumber; // Number of the function 
	fbDebugMsg			: FB_DebugMsg; // Debug Msg Manager (STACK) 
	DebugMsg			: T_MAXSTRING; // Debug msg
	StartTimeMeasurement: T_DCTIME64;	// Get actual time stamp
END_VAR

(**************************************************************************************************************
  Call all emulation functions
***************************************************************************************************************)

// Loop trough all functions 
FOR eFunctionNumber := E_FunctionNumber.F_BEGIN_FUNCTION + 1 TO E_FunctionNumber.F_END_FUNCTION - 1 DO
	// If this function is enabled 
	IF FunctionRegistry[eFunctionNumber].Enable THEN
		// If a valid reference is available 
		IF __ISVALIDREF(FunctionRegistry[eFunctionNumber].rFunction) THEN
			// Start execution time measure
			StartTimeMeasurement := F_GetActualDcTime64();
			// Call
			FunctionRegistry[eFunctionNumber].rFunction();
			
			F_ExecutionTime(
				StartTime			:= StartTimeMeasurement,
				ExecutionTimeSlot 	:= ExecutionTimeTable.Functions[eFunctionNumber]);
		ELSE		
			// Invalid reference
			DebugMsg := CONCAT('F_FunctionComposition - Reference not valid, Function index: ', INT_TO_STRING(eFunctionNumber));
			fbDebugMsg.M_SendErrorMsg(mMessage := DebugMsg);
		END_IF
	END_IF
END_FOR

END_FUNCTION_BLOCK

// ---- 10_Project/10_App/11_Custom/FB_FunctionCompositionCustomized.TcPOU
FUNCTION_BLOCK FB_FunctionCompositionCustomized

fbF_10_001_0200_02_0.CtrlIn.DestinationFunction := F_10_001_0230_01_0;
fbF_10_001_0200_02_0.CtrlIn.DestinationZone := 1;
fbF_10_001_0200_02_0.CtrlIn.TU_Type := 1;

END_FUNCTION_BLOCK

// ---- 20_Product/10_BCF/11_Conv/10_Base/FB_GroupComposition.TcPOU
FUNCTION_BLOCK FB_GroupComposition
(**************************************************************************************
 * 	Application		:	BoxControl Framework
 *	Revision		:	$Revision: 404529 $
 *	Revision date	:	$Date: 2018-04-23 08:21:38 +0200 (Mo., 23 Apr 2018) $
 *	Last changed by	:	$Author: b7bolm $
 *	URL				:	$URL: http://almscdc.swisslog.com/repo/SWPD/Development/BoxControlFramework/20_Release/trunk/01_Software/BCF/BCF/JumpStart/20_Product/10_App/10_Base/10_Lib/10_Conv/FB_GroupComposition.TcPOU $
 *
 *	Purpose			:	Call groups
 *
 * ------------------------------------------------------------------------------------
 *	Copyright Swisslog [IP AG], Switzerland. All rights reserved.
 * 
 * ------------------------------------------------------------------------------------
 *	
 * 	Revision History: 
 *
 * 	VERSION			DATE			INITIALS			DESCRIPTION
 *	0.1				01.01.2001		swl					Example
 *
 **************************************************************************************)
VAR
	eGroupNumber		: E_GroupNumber; // Number of the Group  
	fbDebugMsg			: FB_DebugMsg; // Debug Msg Manager (STACK) 
	DebugMsg			: T_MAXSTRING; // Debug msg
	StartTimeMeasurement: T_DCTIME64;	// Get actual time stamp
END_VAR

(**************************************************************************************************************
  Call all groups
***************************************************************************************************************)
// Loop trough all groups 
FOR eGroupNumber := G_BEGIN_GROUP + 1 TO G_END_GROUP - 1 DO
	// If this group is enabled 
	IF GroupRegistry[eGroupNumber].Enable THEN
		// If a valid reference is available 
		IF __ISVALIDREF(GroupRegistry[eGroupNumber].rGroup) THEN
			// Start execution time measure
			StartTimeMeasurement := F_GetActualDcTime64();
			// Call
			GroupRegistry[eGroupNumber].rGroup();
			
			F_ExecutionTime(
				StartTime			:= StartTimeMeasurement,
				ExecutionTimeSlot 	:= ExecutionTimeTable.Groups[eGroupNumber]);
		ELSE		
			// Invalid reference
			DebugMsg := CONCAT('F_GroupComposition - Reference not valid, Group index: ', INT_TO_STRING(eGroupNumber));
			fbDebugMsg.M_SendErrorMsg(mMessage := DebugMsg);
		END_IF
	END_IF
END_FOR

END_FUNCTION_BLOCK

// ---- 10_Project/10_App/11_Custom/FB_GroupCompositionCustomized.TcPOU
FUNCTION_BLOCK FB_GroupCompositionCustomized


	  //Example of implementation
(*
IF(NOT ProBoxSystem.EMULATION_ENABLED) THEN
	
{region "MONITOR_FUSE_AC"}
	//Group 001
	IF NOT HardwareMapping.I_AK11_FuseAC (* OR NOT HardwareMapping.I_AK11_FuseDC*) THEN 
		// Set error
		F_SetError(	
			ErrorType	:= E_ErrorType.ERROR,
			ErrorParam	:= 'Circuit Break AC AK11 error',
			ErrorMsg	:= E_ErrorConv.CONTROL_VOLTAGE,
			ErrorData	:= Groups.fbSG_001.GroupData.ErrorData.ErrorDataSet[5]);		
	END_IF
		
{endregion}

{region "MONITOR_ASI_BUS"}

	fbSG_001.HW_Inputs.Diag.ASI_BusConfigError						:=AK11_ASI.I.A_1_15.CONF_ERR OR AK11_ASI.I.A_1_15.CONF_ERR;
	fbSG_002.HW_Inputs.Diag.ASI_BusConfigError						:=AK12_ASI.I.A_1_15.CONF_ERR OR AK12_ASI.I.A_1_15.CONF_ERR;
{endregion}

{region "MONITOR_ETHERCAT_DEVICES"}

//	Check IF the Hardware is in the correct state IF NOT the set an error on a group level. Device state 8 = OP, Operational

	//Group 001
	FOR idx := 10 TO 15 DO			 
		 Groups.fbSG_001.M_SetEtherCatError(idx,Subsystem.fbSubsystem.HW_Inputs);		
	END_FOR
	
	//Group 002
	FOR idx := 20 TO 25 DO			 
		 Groups.fbSG_002.M_SetEtherCatError(idx,Subsystem.fbSubsystem.HW_Inputs);		
	END_FOR
	
	//Group 003
	FOR idx := 30 TO 35 DO			 
		 Groups.fbSG_003.M_SetEtherCatError(idx,Subsystem.fbSubsystem.HW_Inputs);		
	END_FOR
		 
{endregion}

END_IF
*)

END_FUNCTION_BLOCK

// ---- 20_Product/10_BCF/11_Conv/10_Base/F_SetError.TcPOU
FUNCTION F_SetError : BOOL
(**************************************************************************************
 * 	Application		:	BoxControl Framework
 *	Revision		:	$Revision: 404529 $
 *	Revision date	:	$Date: 2018-04-23 08:21:38 +0200 (Mo., 23 Apr 2018) $
 *	Last changed by	:	$Author: b7bolm $
 *	URL				:	$URL: http://almscdc.swisslog.com/repo/SWPD/Development/BoxControlFramework/20_Release/trunk/01_Software/BCF/BCF/JumpStart/20_Product/10_App/10_Base/10_Lib/10_Conv/F_SetError.TcPOU $
 *
 *	Purpose			:	Set error
 *						Wrapped to a function to improve debugging and readability.
 *						
 *
 * ------------------------------------------------------------------------------------
 *	Copyright Swisslog [IP AG], Switzerland. All rights reserved.
 * 
 * ------------------------------------------------------------------------------------
 *	
 * 	Revision History: 
 *
 * 	VERSION			DATE			INITIALS			DESCRIPTION
 *	0.1				01.01.2001		swl					Example
 *
 **************************************************************************************)
VAR_INPUT
	ErrorType		: E_ErrorType; // Error message type
	ErrorParam		: STRING(System.ERROR_PARAM_STRINGLENGTH); // Error parameter
	ErrorMsg		: INT; // Error message
END_VAR

VAR_IN_OUT
	ErrorData		: ST_ErrorDataSet; // Error data set
END_VAR

// Check that the values are valid
IF ErrorType > E_ErrorType.NO_ERROR_PENDING AND ErrorMsg > E_ErrorConv.NO_ERROR_CODE THEN
	// Set error
	ErrorData.ErrorType 	:= ErrorType;
	ErrorData.ErrorCode.Conv:= ErrorMsg;
	ErrorData.ErrorParam 	:= ErrorParam;
	
	// Set error successful
	F_SetError 	:= TRUE;
END_IF

END_FUNCTION

// ---- 20_Product/10_BCF/11_Conv/10_Base/FB_SubSystemComposition.TcPOU
FUNCTION_BLOCK FB_SubSystemComposition
(**************************************************************************************
 * 	Application		:	BoxControl Framework
 *	Revision		:	$Revision: 404529 $
 *	Revision date	:	$Date: 2018-04-23 08:21:38 +0200 (Mo., 23 Apr 2018) $
 *	Last changed by	:	$Author: b7bolm $
 *	URL				:	$URL: http://almscdc.swisslog.com/repo/SWPD/Development/BoxControlFramework/20_Release/trunk/01_Software/BCF/BCF/JumpStart/20_Product/10_App/10_Base/10_Lib/10_Conv/FB_SubSystemComposition.TcPOU $
 *
 *	Purpose			:	Call Subsystem 
 *
 * ------------------------------------------------------------------------------------
 *	Copyright Swisslog [IP AG], Switzerland. All rights reserved.
 * 
 * ------------------------------------------------------------------------------------
 *	
 * 	Revision History: 
 *
 * 	VERSION			DATE			INITIALS			DESCRIPTION
 *	0.1				01.01.2001		swl					Example
 *
 **************************************************************************************)
VAR
	fbDebugMsg			: FB_DebugMsg; // Debug Msg Manager (STACK) 
	DebugMsg			: T_MAXSTRING; // Debug msg
	StartTimeMeasurement: T_DCTIME64;	// Get actual time stamp	
END_VAR

(**************************************************************************************************************
   Call the Subsystem manager   
***************************************************************************************************************)

// If a valid reference is available 
IF __ISVALIDREF(SubsystemRegistry.rSubsystem) THEN
	// Start execution time measure
	StartTimeMeasurement := F_GetActualDcTime64();
	// Call 
	SubsystemRegistry.rSubsystem();
	
	F_ExecutionTime(
		StartTime			:= StartTimeMeasurement,
		ExecutionTimeSlot 	:= ExecutionTimeTable.Subsystem);
ELSE		
	// Invalid reference
	DebugMsg := 'F_SubsystemComposition - Reference not valid';
	fbDebugMsg.M_SendErrorMsg(mMessage := DebugMsg);
END_IF

END_FUNCTION_BLOCK

// ---- 10_Project/10_App/11_Custom/FB_SubsystemCompositionCustomized.TcPOU
FUNCTION_BLOCK FB_SubsystemCompositionCustomized


(*
fbPACcapacityCounter(sNetId:= '172.31.5.66.1.1', // enter ams net id of IPC
	                 sFileName:='C:\Users\Test2.csv', // enter user file name and path to crate file automatically
                     LogData01:= F_GetTransportControlData(E_FunctionNumber.F_11_001_0200_01_0,1),
	                 LogData02:= F_GetTransportControlData(E_FunctionNumber.F_11_001_0203_01_0,1));
 *)

END_FUNCTION_BLOCK

// ---- 20_Product/10_BCF/11_Conv/10_Base/FB_DeleteOldTU_Data.TcPOU
FUNCTION_BLOCK FB_DeleteOldTU_Data EXTENDS FB_BaseObject
(**************************************************************************************
 * 	Application		:	BoxControl Framework
 *	Revision		:	$Revision: 404529 $
 *	Revision date	:	$Date: 2018-04-23 08:21:38 +0200 (Mo., 23 Apr 2018) $
 *	Last changed by	:	$Author: b7bolm $
 *	URL				:	$URL: http://almscdc.swisslog.com/repo/SWPD/Development/BoxControlFramework/20_Release/trunk/01_Software/BCF/BCF/JumpStart/20_Product/10_App/10_Base/10_Lib/10_Conv/FB_DeleteOldTU_Data.TcPOU $
 *
 *	Purpose			:	Checks if TU data are expired.
 *
 * ------------------------------------------------------------------------------------
 *	Copyright Swisslog [IP AG], Switzerland. All rights reserved.
 * 
 * ------------------------------------------------------------------------------------
 *	
 * 	Revision History: 
 *
 * VERSION DATE         INITIALS     DESCRIPTION
 * 0.0     DD.MM.YYYY   (name)       (explain customized modifications)
 *
 **************************************************************************************)
VAR
	CurrentDT			: TIMESTRUCT;
	Timespan			: TIME					:= T#0S;
	TU_DataIndex		: DINT					:= 0;		// TU data index
	eFunctionNumber		: E_FunctionNumber		:= 0;		// Function iterator
	Executed			: BOOL					:= FALSE;	// Flag for execution only once
	Position			: ST_PositionIdent;
END_VAR


// Validate every minute all existing TU data
IF fbSystemTime.TIMESTR.wSecond = 0 AND NOT Executed THEN
	// Set execution flag to process only once
	Executed := TRUE;

	// Check 1/60 of the TU data table for old data sets at each execution
	FOR TU_DataIndex := WORD_TO_INT(fbSystemTime.TIMESTR.wMinute) TO NUMBER_OF_TU_DATA BY 60 DO	
		// Check if the TU data set is used 
		IF TU_DataTable[TU_DataIndex].DataSet.DataPresent THEN
			// Delete the TU data set if it is expired 
			CurrentDT:= TU_DataTable[TU_DataIndex].TimeStamp.InsertDateTime;
			Timespan := SYSTEMTIME_TO_DT(System.fbSystemTime.TIMESTR) - SYSTEMTIME_TO_DT(CurrentDT);

			IF (Timespan >= Conveyor.TU_DATA_LIFETIME) THEN
				(*
				Check if this Transport unit is still in use.
				Its possible after holidays that a TU is standing longer than the ExpiryData
				on the system. The time stamp of such units will be updated.
				*)
				Position := F_SearchPositionOfTU_Index(
										TU_DataIndex 		 := TU_DataIndex, 
										eStartFunctionNumber := E_FunctionNumber.F_BEGIN_FUNCTION + 1);
			
				IF Position.eFunctionNumber > E_FunctionNumber.F_BEGIN_FUNCTION THEN
					// Still in use, update time stamp
					TU_DataTable[TU_DataIndex].TimeStamp.InsertDateTime:= System.fbSystemTime.TIMESTR;//TimeStampDT;
				// Otherwise delete data
				ELSE
					// debug message: '11-000-0000-00-0,  expired TU_DataIndex deleted,  TU_DataIndex = 5,  TuID = 000012345,  AssignmentID = 999999999'
					DebugMsg := '';
					DebugMsg := CONCAT(DebugMsg, F_AddDividerToSisString(SubsystemRegistry.SubsystemName));
					DebugMsg := CONCAT(DebugMsg, ',  expired TU_DataIndex deleted');
					DebugMsg := CONCAT(DebugMsg, F_CreateTU_DataString(TU_DataIndex:= TU_DataIndex));
					fbDebugMsg.M_SendErrorMsg(DebugMsg);
					// Loop through all functions 
					F_DeleteTU_Data(
						TU_DataIndex 	:= TU_DataIndex,
						NoTTC 			:= FALSE);
				END_IF
			END_IF
		END_IF
	END_FOR
	
ELSIF fbSystemTime.TIMESTR.wSecond <> 0 THEN
	// Reset execution flag
	Executed := FALSE;
END_IF

END_FUNCTION_BLOCK

// ---- 20_Product/10_BCF/10_Base/FB_BaseObject.TcPOU
FUNCTION_BLOCK FB_BaseObject
(**************************************************************************************
 * 	Application		:	BoxControl Framework
 *	Revision		:	$Revision: 404529 $
 *	Revision date	:	$Date: 2018-04-23 08:21:38 +0200 (Mo., 23 Apr 2018) $
 *	Last changed by	:	$Author: b7bolm $
 *	URL				:	$URL: http://almscdc.swisslog.com/repo/SWPD/Development/BoxControlFramework/20_Release/trunk/01_Software/BCF/BCF/JumpStart/20_Product/10_App/10_Base/10_Lib/FB_BaseObject.TcPOU $
 *
 *	Purpose			:	Base object
 *
 * ------------------------------------------------------------------------------------
 *	Copyright Swisslog [IP AG], Switzerland. All rights reserved.
 * 
 * ------------------------------------------------------------------------------------
 *	
 * 	Revision History: 
 *
 * 	VERSION			DATE			INITIALS			DESCRIPTION
 *	0.1				01.01.2001		swl					Example
 *
 **************************************************************************************)
VAR
	fbDebugMsg		: FB_DebugMsg; // Debug instance
	DebugMsg		: T_MAXSTRING; // Debug msg
	Base			: ST_Base; // Base structure 
END_VAR

(**************************************************************************************************************
   Body never called!
***************************************************************************************************************)
;

METHOD M_ITC_DAQ : BOOL
(**************************************************************************************
 * 	Application		:	BoxControl Framework
 *	Revision		:	$Revision: 404529 $
 *	Revision date	:	$Date: 2018-04-23 08:21:38 +0200 (Mo., 23 Apr 2018) $
 *	Last changed by	:	$Author: b7bolm $
 *	URL				:	$URL: http://almscdc.swisslog.com/repo/SWPD/Development/BoxControlFramework/20_Release/trunk/01_Software/BCF/BCF/JumpStart/20_Product/10_App/10_Base/10_Lib/FB_BaseObject.TcPOU $
 *
 *	Purpose			:	Process incoming DAQ Data Aquisition Request 					
 *
 *
 * ------------------------------------------------------------------------------------
 *	Copyright Swisslog [IP AG], Switzerland. All rights reserved.
 * 
 * ------------------------------------------------------------------------------------
 *	
 * 	Revision History: 
 *
 * 	VERSION			DATE			INITIALS			DESCRIPTION
 *	0.1				01.01.2001		swl					Example
 *
 **************************************************************************************)	
VAR_INPUT
	meChannelSrc		: E_MFCS_CHANNEL; // Number of the source 
	mpData				: PVOID; // Data  pointer 
	mLen				: UDINT; // Data length
END_VAR
(*********************************************************************************
Map Data 	
**********************************************************************************)	
F_BlockCopy(
	pSrc:= mpData, 
	LenSrc:= mLen, 
	pDest:= ADR(Base.CM.DAQ), 
	LenDest:= SIZEOF(Base.CM.DAQ));
// Call Process Method 		
	M_ProcessDAQ(pCM_Data:=ADR(Base.CM),meChannelSrc:= meChannelSrc);
END_METHOD

METHOD M_ITC_DataAquisition : BOOL
(**************************************************************************************
 * 	Application		:	BoxControl Framework
 *	Revision		:	$Revision: 404529 $
 *	Revision date	:	$Date: 2018-04-23 08:21:38 +0200 (Mo., 23 Apr 2018) $
 *	Last changed by	:	$Author: b7bolm $
 *	URL				:	$URL: http://almscdc.swisslog.com/repo/SWPD/Development/BoxControlFramework/20_Release/trunk/01_Software/BCF/BCF/JumpStart/20_Product/10_App/10_Base/10_Lib/FB_BaseObject.TcPOU $
 *
 *	Purpose			:	Method Stores CM Data in Buffer and Sends Report to MFCS when required  					
 *
 *
 * ------------------------------------------------------------------------------------
 *	Copyright Swisslog [IP AG], Switzerland. All rights reserved.
 * 
 * ------------------------------------------------------------------------------------
 *	
 * 	Revision History: 
 *
 * 	VERSION			DATE			INITIALS			DESCRIPTION
 *	0.1				01.01.2001		swl					Example
 *
 **************************************************************************************)	
VAR_INPUT
	mVariableName		: STRING(System.CM_VARIABLENAME_STRINGLENGTH);	///Varaible Name AlphaNumeric string less than 20 Char
	meCM_Index			: E_CM_Index;									/// Index Varaible Storage Array
	mPosition			: STRING(NAME_LENGTH);		///Position Where method is called from
	mCurrentValue		: STRING(Conveyor.GATHERED_DATA_VALUE);			/// Raw data Value to be logged 
	meMode				: E_CM_Mode;									// mode of operation. 
END_VAR
// Call Process Method 	
M_ITC_DataAquisitionProcess(
			mVariableName:= mVariableName, 
			meCM_Index		:= meCM_Index, 
			mPosition		:= mPosition, 
			mCurrentValue	:= mCurrentValue, 
			meMode			:= meMode, 
			pCM_Data		:= ADR(Base.CM));

	M_ITC_DataAquisition:= TRUE;
END_METHOD

METHOD M_ITC_DataAquisitionProcess : BOOL;
(**************************************************************************************
 * 	Application		:	BoxControl Framework
 *	Revision		:	$Revision: 404529 $
 *	Revision date	:	$Date: 2018-04-23 08:21:38 +0200 (Mo., 23 Apr 2018) $
 *	Last changed by	:	$Author: b7bolm $
 *	URL				:	$URL: http://almscdc.swisslog.com/repo/SWPD/Development/BoxControlFramework/20_Release/trunk/01_Software/BCF/BCF/JumpStart/20_Product/10_App/10_Base/10_Lib/FB_BaseObject.TcPOU $
 *
 *	Purpose			:	Method Stores CM Data in Buffer and Sends Report to MFCS when required  					
 *
 *
 * ------------------------------------------------------------------------------------
 *	Copyright Swisslog [IP AG], Switzerland. All rights reserved.
 * 
 * ------------------------------------------------------------------------------------
 *	
 * 	Revision History: 
 *
 * 	VERSION			DATE			INITIALS			DESCRIPTION
 *	0.1				01.01.2001		swl					Example
 *
 **************************************************************************************)	
VAR_INPUT
	mVariableName		: STRING(System.CM_VARIABLENAME_STRINGLENGTH);	///Varaible Name AlphaNumeric string less than 20 Char
	meCM_Index			: E_CM_Index;									/// Index Varaible Storage Array
	mPosition			: STRING(NAME_LENGTH);		///Position Where method is called from
	mCurrentValue		: STRING(Conveyor.GATHERED_DATA_VALUE);			/// Raw data Value to be logged 
	meMode				: E_CM_Mode;									// mode of operation. 
 	pCM_Data			: POINTER TO ST_CM_Base;
END_VAR
VAR
	mCurrentNumValue	: UDINT; // Conversion from String of Sample Value
	mWriteIdx			: INT;	//Temp Write Indes for Buffer 
	mReportSent			: BOOL; //Flag to Check Telegram Sucess
	mEnable				: BOOL; // Enable Logging 
	CycleTime			: TIME;
END_VAR
// Check Input Index is Valid
IF meCM_Index > E_BEGIN_VARIABLE AND 
   meCM_Index < E_END_VARIABLE AND
   pCM_Data <>0 THEN
	
	// Store Variable name
	IF 	pCM_Data^.Settings[meCM_Index].mVariableName <> mVariableName THEN 
		pCM_Data^.Settings[meCM_Index].mVariableName   := mVariableName;
		pCM_Data^.Data[meCM_Index].Position 		   := F_ReduceToAlphaNumeric(mPosition); // Store Position 				
		// Check Mode is Valid 
		IF meMode > E_BEGIN_MODE AND meMode < E_END_MODE THEN
			pCM_Data^.Data[meCM_Index].eMode := meMode;
		ELSE
			pCM_Data^.Data[meCM_Index].eMode := E_CM_Mode.DEFAULT;
		END_IF
 	END_IF;
	
	// Get System Time
	pCM_Data^.nCurrentTime := F_GetCurDcTaskTime64(); // Get current DC-Time (Task-Related)

	//Initialise Max Report Timer
	IF pCM_Data^.Settings[meCM_Index].Enable AND pCM_Data^.Data[meCM_Index].MaxReportTimer = 0 THEN 
		pCM_Data^.Data[meCM_Index].MaxReportTimer		:= pCM_Data^.nCurrentTime + 1000000* TIME_TO_ULINT(pCM_Data^.Settings[meCM_Index].MaxReportTime);
	END_IF;

	
	IF pCM_Data^.Settings[meCM_Index].Enable AND NOT pCM_Data^.Data[meCM_Index].LoggingActive THEN 
		//Logging Started
		pCM_Data^.Data[meCM_Index].LoggingActive := TRUE;
	END_IF;
	
	
	
IF 	pCM_Data^.Data[meCM_Index].LoggingActive THEN 
		// Set Sample time as Cycle time if too low. 
		CycleTime:= DINT_TO_TIME(ActCycleTime/1_000);
		IF pCM_Data^.Settings[meCM_Index].SampleTime < CycleTime THEN
			 pCM_Data^.Settings[meCM_Index].SampleTime := CycleTime;
		END_IF
	
		//Get write Index
		mWriteIdx := pCM_Data^.Data[meCM_Index].WriteIdx;//Temp Write index 
		(*****************************************************************************************************************
		Capture Data 
		******************************************************************************************************************)
			
		
		CASE pCM_Data^.Data[meCM_Index].eMode OF
			(*****************************************************************************************************************
				Value is Alphanumeric 
			******************************************************************************************************************)
			E_CM_Mode.ALPHANUMERIC:  
				 // If Value is a String Value the Threshold value is not used 
				IF  pCM_Data^.nCurrentTime  >= pCM_Data^.Data[meCM_Index].SampleTimer  AND
					pCM_Data^.Data[meCM_Index].WriteIdx <= System.CM_MAX_NUMBER_Of_ENTRIES THEN  
					// Store Sample in Buffer 		
					pCM_Data^.Data[meCM_Index].BUFFER[mWriteIdx].Value  			:= mCurrentValue ;
					pCM_Data^.Data[meCM_Index].BUFFER[mWriteIdx].TimeStamp 		:= LEFT(DCTIME64_TO_STRING(pCM_Data^.nCurrentTime),System.CM_TIMESTAMP_MS_STRINGLENGTH);
					pCM_Data^.Data[meCM_Index].BUFFER[mWriteIdx].Sequence		    := pCM_Data^.Data[meCM_Index].Sequence;			
					pCM_Data^.Data[meCM_Index].WriteIdx							:= pCM_Data^.Data[meCM_Index].WriteIdx + 1;			
				
					// Update Sequence
					IF 	pCM_Data^.Data[meCM_Index].Sequence < 9999 THEN
						pCM_Data^.Data[meCM_Index].Sequence := pCM_Data^.Data[meCM_Index].Sequence+1;
					ELSE
						pCM_Data^.Data[meCM_Index].Sequence := 0;	
					END_IF
					// Reset Sample Time 
					pCM_Data^.Data[meCM_Index].SampleTimer:= pCM_Data^.nCurrentTime +  1000000* TIME_TO_ULINT(pCM_Data^.Settings[meCM_Index].SampleTime);
					
				END_IF;		
		  
			(*****************************************************************************************************************
						Default: Value is a Number
			******************************************************************************************************************)	
	  		E_CM_Mode.DEFAULT:
				mCurrentNumValue := STRING_TO_UDINT(mCurrentValue);//Convert Value to UDINT and copare to +/- Threshold 
				
				IF pCM_Data^.nCurrentTime >= pCM_Data^.Data[meCM_Index].SampleTimer THEN // Check Sampletime 
					// Check Threshold is met
					IF  (	mCurrentNumValue 	>= pCM_Data^.Data[meCM_Index].PreviousValue + INT_TO_UINT(pCM_Data^.Settings[meCM_Index].Threshold) OR 
							mCurrentNumValue	<= pCM_Data^.Data[meCM_Index].PreviousValue - INT_TO_UINT(pCM_Data^.Settings[meCM_Index].Threshold))AND
							pCM_Data^.Data[meCM_Index].WriteIdx <= System.CM_MAX_NUMBER_Of_ENTRIES THEN  
							// Store Sample in Buffer 
							pCM_Data^.Data[meCM_Index].BUFFER[mWriteIdx].Value  			:= UDINT_TO_STRING(mCurrentNumValue) ;
							pCM_Data^.Data[meCM_Index].BUFFER[mWriteIdx].TimeStamp 		:= LEFT(DCTIME64_TO_STRING(pCM_Data^.nCurrentTime),System.CM_TIMESTAMP_MS_STRINGLENGTH);
							pCM_Data^.Data[meCM_Index].BUFFER[mWriteIdx].Sequence		    := pCM_Data^.Data[meCM_Index].Sequence;
							pCM_Data^.Data[meCM_Index].PreviousValue						:= mCurrentNumValue;				
							pCM_Data^.Data[meCM_Index].WriteIdx							:= pCM_Data^.Data[meCM_Index].WriteIdx + 1;
							
							// Update Sequence 
							IF 	pCM_Data^.Data[meCM_Index].Sequence < 9999 THEN
								pCM_Data^.Data[meCM_Index].Sequence	:= pCM_Data^.Data[meCM_Index].Sequence+1;
							ELSE
								pCM_Data^.Data[meCM_Index].Sequence 	:= 0;	
							END_IF
					END_IF;
					// Reset Sample Time 
					pCM_Data^.Data[meCM_Index].SampleTimer:= pCM_Data^.nCurrentTime +  1000000* TIME_TO_ULINT(pCM_Data^.Settings[meCM_Index].SampleTime);
				END_IF;
		END_CASE

		(**********************************************************************************************************************
		Send Report If Requested 
		************************************************************************************************************************)
		mReportSent := FALSE;
	
		IF   (pCM_Data^.nCurrentTime >= pCM_Data^.Data[meCM_Index].MaxReportTimer) AND //Max Report Time is Reached
			 (pCM_Data^.Data[meCM_Index].MaxReportTimer >0) AND
			 (pCM_Data^.Settings[meCM_Index].MaxReportTime>T#0MS)OR
			  pCM_Data^.Data[meCM_Index].WriteIdx >= System.CM_MAX_NUMBER_Of_ENTRIES AND // Buffer is full 
			  pCM_Data^.Data[meCM_Index].WriteIdx >0  THEN 
			//Send Report.
			mReportSent:=  F_ITC_SendGDR(
								eChannelSrc			:= E_MFCS_Channel.CM, 
								Position			:= pCM_Data^.Data[meCM_Index].Position,
								Variable			:= pCM_Data^.Settings[meCM_Index].mVariableName,
								NumberOfSets		:= pCM_Data^.Data[meCM_Index].WriteIdx, 
								DataSet				:= pCM_Data^.Data[meCM_Index].BUFFER, 
								eReturnCode			:= 0);
				 
				//Check if Report Failed to Send
				IF NOT mReportSent AND NOT pCM_Data^.Settings[meCM_Index].Option THEN
						pCM_Data^.Settings[meCM_Index].Enable := FALSE;
						pCM_Data^.Settings[meCM_Index].ErrorCode := 1000;
						F_ITC_SendDAR(
							eChannelSrc		:= E_MFCS_Channel.CM , 
							Position		:= pCM_Data^.Data[meCM_Index].Position, 
							Code			:= 0, 
							NumberOfSets	:= 1, 
							SET				:= pCM_Data^.Settings, 
							SetOffset		:= meCM_Index,
							eErrorCode		:= 0 );	
				END_IF
			// Reset Max Report Time 	
			 pCM_Data^.Data[meCM_Index].WriteIdx  			:= 0;// Reset Write Index after Report Sent.
			 pCM_Data^.Data[meCM_Index].MaxReportTimer		:= pCM_Data^.nCurrentTime + 1000000* TIME_TO_ULINT(pCM_Data^.Settings[meCM_Index].MaxReportTime);

		ELSIF NOT pCM_Data^.Settings[meCM_Index].Enable THEN // Stop logging Request from user. 
			//Send Report.
			mReportSent:=  F_ITC_SendGDR(
								eChannelSrc				:= E_MFCS_Channel.CM, 
								Position				:= pCM_Data^.Data[meCM_Index].Position,
								Variable				:= pCM_Data^.Settings[meCM_Index].mVariableName,
								NumberOfSets			:= pCM_Data^.Data[meCM_Index].WriteIdx, 
								DataSet					:= pCM_Data^.Data[meCM_Index].BUFFER, 
								eReturnCode				:= 0);			
			// Reset
			 pCM_Data^.Data[meCM_Index].WriteIdx  			:= 0;// Reset Write Index after Report Sent.
			 pCM_Data^.Data[meCM_Index].MaxReportTimer		:= 0; // Reset Max Report Timer 
			 pCM_Data^.Data[meCM_Index].Sequence 			:= 0; // Reset Sequence 
			 pCM_Data^.Data[meCM_Index].SampleTimer 		:= 0; // Reset Sample timer 
			 pCM_Data^.Data[meCM_Index].PreviousValue		:= 0; // Reset Last Value Logged
			 pCM_Data^.Data[meCM_Index].LoggingActive 		:= FALSE;	 // Turn off Logging.
		END_IF
	END_IF;	
END_IF

M_ITC_DataAquisitionProcess := TRUE;
END_METHOD

METHOD M_ITC_GDQ : BOOL
(**************************************************************************************
 * 	Application		:	BoxControl Framework
 *	Revision		:	$Revision: 404529 $
 *	Revision date	:	$Date: 2018-04-23 08:21:38 +0200 (Mo., 23 Apr 2018) $
 *	Last changed by	:	$Author: b7bolm $
 *	URL				:	$URL: http://almscdc.swisslog.com/repo/SWPD/Development/BoxControlFramework/20_Release/trunk/01_Software/BCF/BCF/JumpStart/20_Product/10_App/10_Base/10_Lib/FB_BaseObject.TcPOU $
 *
 *	Purpose			:	Process incoming GDQ Gathered Data Request 					
 *
 *
 * ------------------------------------------------------------------------------------
 *	Copyright Swisslog [IP AG], Switzerland. All rights reserved.
 * 
 * ------------------------------------------------------------------------------------
 *	
 * 	Revision History: 
 *
 * 	VERSION			DATE			INITIALS			DESCRIPTION
 *	0.1				01.01.2001		swl					Example
 *
 **************************************************************************************)	
VAR_INPUT
	meChannelSrc		: E_MFCS_CHANNEL; // Number of the source 
	mpData				: PVOID; // Data  pointer 
	mLen				: UDINT; // Data length
END_VAR
// Map data
F_BlockCopy(
	pSrc:= mpData, 
	LenSrc:= mLen, 
	pDest:= ADR(Base.CM.GDQ), 
	LenDest:= SIZEOF(Base.CM.GDQ));
// Call Process Method 	
	M_ProcessGDQ(pCM_Data:=ADR(Base.CM),meChannelSrc := meChannelSrc);
END_METHOD

METHOD M_ITC_ProcessMsg : BOOL
VAR_INPUT
	meChannelSrc		: E_MFCS_CHANNEL; // Number of the source 
	mMsgType			: INT; // Message type
	mpData				: PVOID; // Data  pointer 
	mLen				: UDINT; // Data length
END_VAR
(*
This method serves as dummy to fullfil interface requirements.

This is needed to keep independency between library product types.

This method should be overwriten in each Rootclass underneath.

*)
END_METHOD

METHOD PROTECTED M_ITC_VIQ : BOOL
(**************************************************************************************
 * 	Application		:	BoxControl Framework
 *	Revision		:	$Revision: 404529 $
 *	Revision date	:	$Date: 2018-04-23 08:21:38 +0200 (Mo., 23 Apr 2018) $
 *	Last changed by	:	$Author: b7bolm $
 *	URL				:	$URL: http://almscdc.swisslog.com/repo/SWPD/Development/BoxControlFramework/20_Release/trunk/01_Software/BCF/BCF/JumpStart/20_Product/10_App/10_Base/10_Lib/FB_BaseObject.TcPOU $
 *
 *	Purpose			:	Process incoming VIQ - Visualization Info Request
 *
 * ------------------------------------------------------------------------------------
 *	Copyright Swisslog [IP AG], Switzerland. All rights reserved.
 * 
 * ------------------------------------------------------------------------------------
 *	
 * 	Revision History: 
 *
 * 	VERSION			DATE			INITIALS			DESCRIPTION
 *	0.1				01.01.2001		swl					Example
 *
 **************************************************************************************)
VAR_INPUT
	meChannelSrc		: E_MFCS_CHANNEL; // Number of the source 
	mpData				: PVOID; // Data  pointer 
	mLen				: UDINT; // Data length
END_VAR

VAR
	mIdx,mIdx2			: INT; // Iterator
	mCompString1		: STRING(System.KEY_LENGTH);
	mCompString2		: STRING(System.KEY_LENGTH);
	mNumberOfUsedKeys	: INT; 
END_VAR
// Initialize 
M_ITC_VIQ := TRUE;

// Map data
F_BlockCopy(
	pSrc:= mpData, 
	LenSrc:= mLen, 
	pDest:= ADR(Base.VIQ), 
	LenDest:= SIZEOF(Base.VIQ));

// Clear preparation data struct
MEMSET(destAddr := ADR(Base.VIR_Data.PrepData), fillByte := 0, n := SIZEOF(Base.VIR_Data.PrepData));

(*
If all used variables were requested
NumberOfKeys = 0
*)
IF Base.VIQ.NumberOfKeys = 0 THEN
	// Send all used (Notified by M_VIR_Update)
	mNumberOfUsedKeys := Base.VIR_Data.NumberOfUsedKeys;
	Base.VIR_Data.PrepData := Base.VIR_Data.Data;
	
(*
Otherwise only specific keys were requested.
Search and report them.
*)
ELSE
	mNumberOfUsedKeys := Base.VIQ.NumberOfKeys;
	FOR mIdx := 1 TO mNumberOfUsedKeys BY 1 DO
		// Store search key and search
		Base.VIR_Data.PrepData[mIdx].Key := Base.VIQ.Keys[mIdx];	
	
		FOR mIdx2 := 1 TO System.NUMBER_OF_KEYVALUE_PAIRS_VIR DO
			(* 
			Prepare string to compare - Remove blanks, all to upper case
			*)
			mCompString1 := F_ToUCase(F_ReduceToAlphaNumeric(InputString:= Base.VIQ.Keys[mIdx]));
			mCompString2 := F_ToUCase(Base.VIR_Data.Data[mIdx2].Key);
			// If a key matches store current value otherwise -1 to inform key not found
			IF mCompString1 = mCompString2 THEN
				Base.VIR_Data.PrepData[mIdx].Value := Base.VIR_Data.Data[mIdx2].Value;
				EXIT;
			ELSIF mIdx2 >= System.NUMBER_OF_KEYVALUE_PAIRS_VIR THEN
				Base.VIR_Data.PrepData[mIdx].Value := '-1';
			END_IF
		END_FOR
	END_FOR
END_IF

// Send report
F_ITC_SendVIR(
	eChannelSrc	:= E_MFCS_Channel.SPOC,
	Position := F_ReduceToAlphaNumeric(Base.VIQ.Position),
	NumOfKeyValuePairs := mNumberOfUsedKeys,
	KeyValuePairs := Base.VIR_Data.PrepData);
END_METHOD

METHOD M_ProcessDAQ : BOOL
(**************************************************************************************
 * 	Application		:	BoxControl Framework
 *	Revision		:	$Revision: 404529 $
 *	Revision date	:	$Date: 2018-04-23 08:21:38 +0200 (Mo., 23 Apr 2018) $
 *	Last changed by	:	$Author: b7bolm $
 *	URL				:	$URL: http://almscdc.swisslog.com/repo/SWPD/Development/BoxControlFramework/20_Release/trunk/01_Software/BCF/BCF/JumpStart/20_Product/10_App/10_Base/10_Lib/FB_BaseObject.TcPOU $
 *
 *	Purpose			:	Process incoming DAQ Data Aquisition Request 					
 *
 *
 * ------------------------------------------------------------------------------------
 *	Copyright Swisslog [IP AG], Switzerland. All rights reserved.
 * 
 * ------------------------------------------------------------------------------------
 *	
 * 	Revision History: 
 *
 * 	VERSION			DATE			INITIALS			DESCRIPTION
 *	0.1				01.01.2001		swl					Example
 *
 **************************************************************************************)	
VAR_INPUT
	meChannelSrc		: E_MFCS_CHANNEL; // Number of the source 
 	pCM_Data			: POINTER TO ST_CM_Base;
END_VAR
VAR
	mCompString1		: STRING(System.CM_VARIABLENAME_STRINGLENGTH);
	mCompString2		: STRING(System.CM_VARIABLENAME_STRINGLENGTH);
	meCM_Index			: E_CM_Index;	/// Index Data Storage Array
	mIdx2				: INT; //Iterator 
END_VAR

(*********************************************************************************
Switch OF ALL Logging if Requested. 	
**********************************************************************************)	
IF pCM_Data^.DAQ.Code = 1 THEN
	FOR meCM_Index:= E_BEGIN_VARIABLE+1 TO E_END_VARIABLE -1 DO 
		IF pCM_Data^.Settings[meCM_Index].Enable THEN
			pCM_Data^.Settings[meCM_Index].Enable := FALSE; // Turn Off Logging 
		END_IF;
	END_FOR
END_IF


(*********************************************************************************	
Process Sets Data 
**********************************************************************************)	
IF  pCM_Data^.DAQ.NumberOfSets >0 AND pCM_Data^.DAQ.Code = 0 THEN	//Telegram contains "Set" Parameters 	 
	FOR	mIdx2:= 1 TO pCM_Data^.DAQ.NumberOfSets 	DO				//Itereate though Recieved Telgram Sets
		FOR meCM_Index:= E_BEGIN_VARIABLE+1 TO E_END_VARIABLE -1 DO // Iterate through Stored PLC data 
			mCompString1:= F_ToUCase(F_ReduceToAlphaNumeric(pCM_Data^.Settings[meCM_Index].mVariableName));
			mCompString2:= F_ToUCase(F_ReduceToAlphaNumeric(pCM_Data^.DAQ.Set[mIdx2].mVariableName));
			IF mCompString1 = mCompString2 THEN 
				 pCM_Data^.Settings[meCM_Index]		:= pCM_Data^.DAQ.Set[mIdx2]; // Write Data to Storage location 
			END_IF			
		END_FOR;	
	END_FOR;
END_IF;

(*********************************************************************************
Send Data Aquisitiion Report
**********************************************************************************)	
FOR meCM_Index:= E_BEGIN_VARIABLE+1 TO E_END_VARIABLE -1 DO 
	IF	pCM_Data^.Settings[meCM_Index].mVariableName =''  THEN 
		EXIT;
	END_IF	
END_FOR;

F_ITC_SendDAR(
			eChannelSrc		:= meChannelSrc, 
			Position		:= pCM_Data^.DAQ.Position, 
			Code			:= pCM_Data^.DAQ.Code, 
			NumberOfSets	:= meCM_Index-1, 
			SET				:= pCM_Data^.Settings, 
			SetOffset		:= E_CM_Index.E_BEGIN_VARIABLE,
			eErrorCode		:= E_ErrorConv.NO_ERROR_CODE );
END_METHOD

METHOD M_ProcessGDQ : BOOL
(**************************************************************************************
 * 	Application		:	BoxControl Framework
 *	Revision		:	$Revision: 404529 $
 *	Revision date	:	$Date: 2018-04-23 08:21:38 +0200 (Mo., 23 Apr 2018) $
 *	Last changed by	:	$Author: b7bolm $
 *	URL				:	$URL: http://almscdc.swisslog.com/repo/SWPD/Development/BoxControlFramework/20_Release/trunk/01_Software/BCF/BCF/JumpStart/20_Product/10_App/10_Base/10_Lib/FB_BaseObject.TcPOU $
 *
 *	Purpose			:	Process incoming GDQ Gathered Data Request 					
 *
 *
 * ------------------------------------------------------------------------------------
 *	Copyright Swisslog [IP AG], Switzerland. All rights reserved.
 * 
 * ------------------------------------------------------------------------------------
 *	
 * 	Revision History: 
 *
 * 	VERSION			DATE			INITIALS			DESCRIPTION
 *	0.1				01.01.2001		swl					Example
 *
 **************************************************************************************)	
VAR_INPUT
	meChannelSrc		: E_MFCS_CHANNEL; // Number of the source 
 	pCM_Data			: POINTER TO ST_CM_Base;
END_VAR
VAR
	mCompString1		: STRING(System.CM_VARIABLENAME_STRINGLENGTH);
	mCompString2		: STRING(System.CM_VARIABLENAME_STRINGLENGTH);
	meCM_Index			: E_CM_Index;/// Index Data Storage Array
	mReportSent			: BOOL;	//Flag to Check Telegram Sucess
END_VAR
	
mReportSent  := FALSE;
(*********************************************************************************	
Process Telegram
**********************************************************************************)	
FOR meCM_Index:= E_BEGIN_VARIABLE+1 TO E_END_VARIABLE -1 DO  //Iterate through PLC Storage location
	mCompString1:= F_ToUCase(F_ReduceToAlphaNumeric(pCM_Data^.Settings[meCM_Index].mVariableName));
	mCompString2:= F_ToUCase(F_ReduceToAlphaNumeric(pCM_Data^.GDQ.Variable));
	IF mCompString1 = mCompString2 AND // Compare Names 
		pCM_Data^.Data[meCM_Index].LoggingActive THEN 
		// Send Gathered Data Report 
		mReportSent:=  F_ITC_SendGDR(
									eChannelSrc				:= meChannelSrc, 
									Position				:= pCM_Data^.Data[meCM_Index].Position,
									Variable				:= pCM_Data^.Settings[meCM_Index].mVariableName,
									NumberOfSets			:= pCM_Data^.Data[meCM_Index].WriteIdx, 
									DataSet					:= pCM_Data^.Data[meCM_Index].BUFFER, 
									eReturnCode				:= 0);				
							
		//Check if Report Failed to Send
		IF NOT mReportSent AND NOT Base.CM.Settings[meCM_Index].Option THEN
			pCM_Data^.Settings[meCM_Index].Enable := FALSE; //  Reset Enable 
			pCM_Data^.Settings[meCM_Index].ErrorCode := 1000;
			//Send Report with Error Code.
			F_ITC_SendDAR(
								eChannelSrc		:= meChannelSrc , 
								Position		:= pCM_Data^.Data[meCM_Index].Position, 
								Code			:= 0, 
								NumberOfSets	:= 1, 
								SET				:= pCM_Data^.Settings, 
								SetOffset		:= meCM_Index,
								eErrorCode		:= 0 );																									
		END_IF
		
		// Update Index and Timer
		pCM_Data^.Data[meCM_Index].WriteIdx  			:= 0;// Reset Write Index after Report Sent.
		pCM_Data^.Data[meCM_Index].MaxReportTimer		:= pCM_Data^.nCurrentTime + 1000000* TIME_TO_ULINT(pCM_Data^.Settings[meCM_Index].MaxReportTime);
		EXIT;											
	END_IF;
END_FOR
END_METHOD

METHOD M_VIR_Update : BOOL
(**************************************************************************************
 * 	Application		:	BoxControl Framework
 *	Revision		:	$Revision: 404529 $
 *	Revision date	:	$Date: 2018-04-23 08:21:38 +0200 (Mo., 23 Apr 2018) $
 *	Last changed by	:	$Author: b7bolm $
 *	URL				:	$URL: http://almscdc.swisslog.com/repo/SWPD/Development/BoxControlFramework/20_Release/trunk/01_Software/BCF/BCF/JumpStart/20_Product/10_App/10_Base/10_Lib/FB_BaseObject.TcPOU $
 *
 *	Purpose			:	Update Visualization report.
 *						This method controls sending of viszualization reports.
 *						A report will be sent if a data change happened and its 
 *						allowed to send a new report. 
 *						As a reason that this is a visualization report - the allowed
 *						sending intervall is limited hard coded.
 *						This Method needs to be called if VIR/VIQ are requested.
 *
 * ------------------------------------------------------------------------------------
 *	Copyright Swisslog [IP AG], Switzerland. All rights reserved.
 * 
 * ------------------------------------------------------------------------------------
 *	
 * 	Revision History: 
 *
 * 	VERSION			DATE			INITIALS			DESCRIPTION
 *	0.1				01.01.2001		swl					Example
 *
 **************************************************************************************)
VAR_INPUT
	mPosition			: STRING(System.NAME_LENGTH); // Position name
	mNumberOfValues		: INT; // Number of used values 
END_VAR
// Init
M_VIR_Update := FALSE;

Base.VIR_Data.NumberOfUsedKeys := mNumberOfValues;

// Validate inputs
IF mNumberOfValues > 0 AND
   mNumberOfValues <= System.NUMBER_OF_KEYVALUE_PAIRS_VIR THEN

	// Update current system time
	Base.fbGetSystemTime();
	
	IF NOT Base.VIR_Data.SendingAllowed THEN
		IF Base.VIR_Data.Overflow THEN
			// Wait until its allowed to send a new request
			IF Base.fbGetSystemTime.timeLoDW - 4294967296 > Base.VIR_Data.NextSendTimeStamp THEN
				Base.VIR_Data.SendingAllowed := TRUE;
				Base.VIR_Data.Overflow := FALSE;
			END_IF
		// Wait until its allowed to send a new request
		ELSIF Base.fbGetSystemTime.timeLoDW > Base.VIR_Data.NextSendTimeStamp THEN
			Base.VIR_Data.SendingAllowed := TRUE;
		END_IF
	ELSE
		// Only send if change was detected
		IF Base.VIR_Data.ChangeDetected THEN
			// Send report
			F_ITC_SendVIR(
				eChannelSrc	:= 0, 
				Position:= F_ReduceToAlphaNumeric(mPosition), 
				NumOfKeyValuePairs:= mNumberOfValues, 
				KeyValuePairs:= Base.VIR_Data.Data);
				
			// Reset values
			Base.VIR_Data.ChangeDetected := FALSE;
			Base.VIR_Data.SendingAllowed := FALSE;
			
			// Calculate next time stamp
			Base.VIR_Data.TimeStep := Base.VIR_SEND_CLOCK * 10000000;
			Base.VIR_Data.NextSendTimeStamp := Base.fbGetSystemTime.timeLoDW + Base.VIR_Data.TimeStep;
		
			IF Base.VIR_Data.NextSendTimeStamp < Base.fbGetSystemTime.timeLoDW THEN
				Base.VIR_Data.Overflow := TRUE;
			END_IF
		END_IF
	END_IF
	
	// Process successful
	M_VIR_Update := TRUE;
END_IF
END_METHOD

METHOD M_VIR_Value : BOOL
(**************************************************************************************
 * 	Application		:	BoxControl Framework
 *	Revision		:	$Revision: 404529 $
 *	Revision date	:	$Date: 2018-04-23 08:21:38 +0200 (Mo., 23 Apr 2018) $
 *	Last changed by	:	$Author: b7bolm $
 *	URL				:	$URL: http://almscdc.swisslog.com/repo/SWPD/Development/BoxControlFramework/20_Release/trunk/01_Software/BCF/BCF/JumpStart/20_Product/10_App/10_Base/10_Lib/FB_BaseObject.TcPOU $
 *
 *	Purpose			:	Update Visualization report.
 *						This method is used to handle a variable which needs to be reported
 *						by visualization report.
 *						This method handles only recording - method M_VIR_Update needs
 *						to be called to handle the communication.					
 *
 *
 * ------------------------------------------------------------------------------------
 *	Copyright Swisslog [IP AG], Switzerland. All rights reserved.
 * 
 * ------------------------------------------------------------------------------------
 *	
 * 	Revision History: 
 *
 * 	VERSION			DATE			INITIALS			DESCRIPTION
 *	0.1				01.01.2001		swl					Example
 *
 **************************************************************************************)
VAR_INPUT
	mIndex			: INT; // Used Index
	mKey			: STRING(System.KEY_LENGTH); // Key for value
	mValue			: STRING(System.VALUE_LENGTH); // Current Value as String
	mEventTrigger	: BOOL; // Request on value change (Otherwise polling over VIQ)
END_VAR
// Init
M_VIR_Value := FALSE;

// Validate inputs
IF mIndex > 0 AND
   mIndex <= System.NUMBER_OF_KEYVALUE_PAIRS_VIR AND
   LEN(mKey) > 0 AND
   LEN(mValue) > 0 THEN
   // Store key
   	Base.VIR_Data.Data[mIndex].Key := mKey;

	// Compare value
	IF MEMCMP(ADR(mValue), ADR(Base.VIR_Data.Data[mIndex].Value),INT_TO_UDINT(LEN(Base.VIR_Data.Data[mIndex].Value))) <> 0 OR 
       LEN(Base.VIR_Data.Data[mIndex].Value) <> LEN(mValue) THEN
		// Update value, set flag for report
		Base.VIR_Data.Data[mIndex].Value := mValue;
		
		// Mark change
		IF NOT Base.VIR_Data.ChangeDetected THEN
			Base.VIR_Data.ChangeDetected := mEventTrigger;
		END_IF
	END_IF

	// Process successful
	M_VIR_Value := TRUE;
END_IF
END_METHOD

END_FUNCTION_BLOCK

// ---- 20_Product/30_Toolbox/12_StringStream/F_ReduceToAlphaNumeric.TcPOU
FUNCTION F_ReduceToAlphaNumeric : STRING(255)
(**************************************************************************************
 * 	Application		:	BoxControl Framework
 *	Revision		:	$Revision: 404529 $
 *	Revision date	:	$Date: 2018-04-23 08:21:38 +0200 (Mo., 23 Apr 2018) $
 *	Last changed by	:	$Author: b7bolm $
 *	URL				:	$URL: http://almscdc.swisslog.com/repo/SWPD/Development/BoxControlFramework/20_Release/trunk/01_Software/BCF/BCF/JumpStart/30_Toolbox/12_StringStream/F_ReduceToAlphaNumeric.TcPOU $
 *
 *	Purpose			:	Remove non alpha numeric signs from a string.
 *
 * ------------------------------------------------------------------------------------
 *	Copyright Swisslog [IP AG], Switzerland. All rights reserved.
 * 
 * ------------------------------------------------------------------------------------
 *	
 * 	Revision History: 
 *
 * 	VERSION			DATE			INITIALS			DESCRIPTION
 *	0.1				01.01.2001		swl					Example
 *
 **************************************************************************************)
VAR_INPUT
	InputString		: STRING(255); // Input string
END_VAR
VAR
	Idx				: INT; // Iterator
	pASCII_Array	: POINTER TO ARRAY[1..255] OF BYTE;
	ASCII_Value		: INT; // Value
END_VAR

// Initialize
F_ReduceToAlphaNumeric := '';

// Build ASCII array
pASCII_Array := ADR(InputString);

// Go Through string
FOR Idx := 1 TO LEN(InputString) DO
	// Get first ASCII sign as INT
	ASCII_Value := BYTE_TO_INT(pASCII_Array^[Idx]);
	
	// Only if it is a char between 0..9, A..Z, a..z 
	IF  ((ASCII_Value > 47) AND (ASCII_Value < 58)) OR
	 	((ASCII_Value > 64) AND (ASCII_Value < 91)) OR
	 	((ASCII_Value > 96) AND (ASCII_Value < 123)) THEN
		
		// Build string
		fbFormatString( sFormat := '%C',
						arg1 	:= F_BYTE(pASCII_Array^[Idx]));
		
		// Return alpha numeric string
		F_ReduceToAlphaNumeric := CONCAT(F_ReduceToAlphaNumeric, fbFormatString.sOut);
	END_IF
END_FOR

END_FUNCTION

// ---- 20_Product/10_BCF/11_Conv/11_Com/11_ITC/F_ITC_SendGDR.TcPOU
FUNCTION F_ITC_SendGDR : BOOL
(**************************************************************************************
 * 	Application		:	BoxControl Framework
 *	Revision		:	$Revision: 404529 $
 *	Revision date	:	$Date: 2018-04-23 08:21:38 +0200 (Mo., 23 Apr 2018) $
 *	Last changed by	:	$Author: b7bolm $
 *	URL				:	$URL: http://almscdc.swisslog.com/repo/SWPD/Development/BoxControlFramework/20_Release/trunk/01_Software/BCF/BCF/JumpStart/20_Product/10_App/11_Com/10_Lib/10_Conv/11_ITC/F_ITC_SendGDR.TcPOU $
 *
 *	Purpose			:	Wrap message - GDR					
 *
 *
 * ------------------------------------------------------------------------------------
 *	Copyright Swisslog [IP AG], Switzerland. All rights reserved.
 * 
 * ------------------------------------------------------------------------------------
 *	
 * 	Revision History: 
 *
 * 	VERSION			DATE			INITIALS			DESCRIPTION
 *	0.1				01.01.2001		swl					Example
 *
 **************************************************************************************)	
VAR_INPUT
	eChannelSrc		: E_MFCS_Channel;/// Source communicaton channel	
	Position		: STRING(Conveyor.POSITION_STRINGLENGTH);// SIS Group Name MM-GGG-0000-000
	Variable		: STRING(System.CM_VARIABLE_STRINGLENGTH);// Variable Name
	NumberOfSets	: INT;// Number of data captures to be proccessed 
	DataSet			: ARRAY[0..System.CM_MAX_NUMBER_Of_ENTRIES] OF ST_CM_LOG; //Data 
	eReturnCode		: E_ErrorConv;	/// Return code
END_VAR
VAR
	GDR				: ST_ITC_GDR; //Gathered Data Report Structure
END_VAR

// Map values
GDR.Position 		:= Position;
GDR.Variable 		:= Variable;
GDR.NumberOfSets 	:= NumberOfSets;
GDR.DataSet			:= DataSet;
GDR.eReturnCode  	:= eReturnCode;

// Forward to ITC
F_ITC_SendGDR := fbITC_Manager.M_SendData(
					meChannel	:= eChannelSrc,
					mMsgType	:= E_ITC_MsgTypeConv.GATHERED_DATA_REPORT,
					mpData		:= ADR(GDR),
					mLen		:= SIZEOF(GDR));

END_FUNCTION

// ---- 20_Product/10_BCF/11_Conv/11_Com/11_ITC/F_ITC_SendDAR.TcPOU
FUNCTION F_ITC_SendDAR : BOOL
(**************************************************************************************
 * 	Application		:	BoxControl Framework
 *	Revision		:	$Revision: 404529 $
 *	Revision date	:	$Date: 2018-04-23 08:21:38 +0200 (Mo., 23 Apr 2018) $
 *	Last changed by	:	$Author: b7bolm $
 *	URL				:	$URL: http://almscdc.swisslog.com/repo/SWPD/Development/BoxControlFramework/20_Release/trunk/01_Software/BCF/BCF/JumpStart/20_Product/10_App/11_Com/10_Lib/10_Conv/11_ITC/F_ITC_SendDAR.TcPOU $
 *
 *	Purpose			:	Wrap message - DAR
 *
 * ------------------------------------------------------------------------------------
 *	Copyright Swisslog [IP AG], Switzerland. All rights reserved.
 * 
 * ------------------------------------------------------------------------------------
 *	
 * 	Revision History: 
 *
 * 	VERSION			DATE			INITIALS			DESCRIPTION
 *	0.1				01.01.2001		swl					Example
 *
 **************************************************************************************)
VAR_INPUT
	eChannelSrc			: E_MFCS_Channel;	/// Source communicaton channel	
	Position			: STRING(Conveyor.POSITION_STRINGLENGTH);// SIS MM-GGG-EEEE-FF-Z
	Code				: INT; //Request = 0 Off ALL = 1
	NumberOfSets		: INT; // Number of Sets to be Proccessed in Telegram
	Set					: ARRAY[E_CM_Index.E_BEGIN_VARIABLE+1..E_CM_Index.E_END_VARIABLE-1] OF ST_CM_Settings;
	SetOffset			: E_CM_Index; // Set Offset if less than all availble sets are sent
	eErrorCode			: E_ErrorConv; // Error Code 
END_VAR
VAR
	DAR					: ST_ITC_DAR; //Data Aquisiiton Report Structure 
END_VAR

// Map values  	
DAR.Position		:= Position;
DAR.Code			:= Code;
DAR.NumberOfSets 	:= NumberOfSets;
DAR.Set				:= Set;
DAR.SetOffset		:= SetOffset;
DAR.eErrorCode		:= eErrorcode;
// Forward to ITC	
F_ITC_SendDAR := fbITC_Manager.M_SendData(
					meChannel	:= eChannelSrc,
					mMsgType	:= E_ITC_MsgTypeConv.DATA_ACQUISITION_REPORT,
					mpData		:= ADR(DAR),
					mLen		:= SIZEOF(DAR));

END_FUNCTION

// ---- 20_Product/10_BCF/10_Base/11_Com/F_ITC_SendVIR.TcPOU
FUNCTION F_ITC_SendVIR : BOOL
(**************************************************************************************
 * 	Application		:	BoxControl Framework
 *	Revision		:	$Revision: 404529 $
 *	Revision date	:	$Date: 2018-04-23 08:21:38 +0200 (Mo., 23 Apr 2018) $
 *	Last changed by	:	$Author: b7bolm $
 *	URL				:	$URL: http://almscdc.swisslog.com/repo/SWPD/Development/BoxControlFramework/20_Release/trunk/01_Software/BCF/BCF/JumpStart/20_Product/10_App/11_Com/10_Lib/F_ITC_SendVIR.TcPOU $
 *
 *	Purpose			:	Wrap message - POR
 *
 * ------------------------------------------------------------------------------------
 *	Copyright Swisslog [IP AG], Switzerland. All rights reserved.
 * 
 * ------------------------------------------------------------------------------------
 *	
 * 	Revision History: 
 *
 * 	VERSION			DATE			INITIALS			DESCRIPTION
 *	0.1				01.01.2001		swl					Example
 *
 **************************************************************************************)
VAR_INPUT
	eChannelSrc			: E_MFCS_Channel; // Source communicaton channel		
	Position			: STRING(System.NAME_LENGTH); // SIS MM-GGG-EEEE-FF-Z
	NumOfKeyValuePairs	: INT;
	KeyValuePairs		: ARRAY [1..System.NUMBER_OF_KEYVALUE_PAIRS_VIR] OF ST_ITC_VIR_SET;
END_VAR
VAR
	VIR					: ST_ITC_VIR;
	Idx					: INT; 
END_VAR

